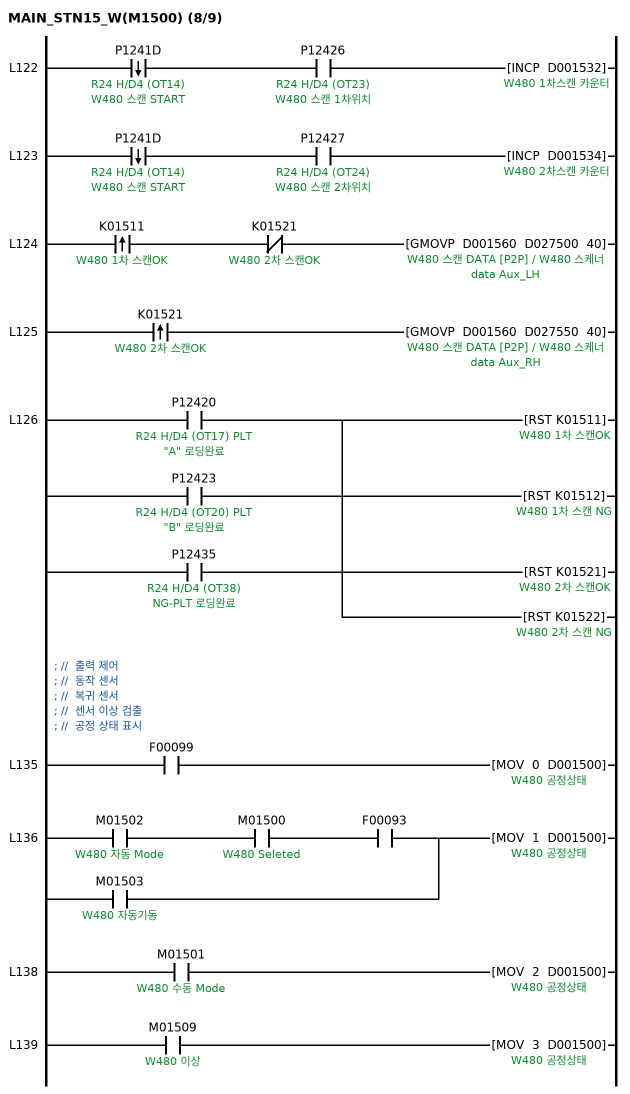
[picture p240: MAIN_STN15_W(M1500) rungs L122-L139]
; L122
LOADN     P1241D	// R24 H/D4 (OT14) W480 스캔 START
AND       P12426	// R24 H/D4 (OT23) W480 스캔 1차위치
INCP      D001532	// W480 1차스캔 카운터
; L123
LOADN     P1241D	// R24 H/D4 (OT14) W480 스캔 START
AND       P12427	// R24 H/D4 (OT24) W480 스캔 2차위치
INCP      D001534	// W480 2차스캔 카운터
; L124
LOADP     K01511	// W480 1차 스캔OK
AND NOT   K01521	// W480 2차 스캔OK
GMOVP     D001560 D027500 40	// W480 스캔 DATA [P2P] / W480 스케너 data Aux_LH
; L125
LOADP     K01521	// W480 2차 스캔OK
GMOVP     D001560 D027550 40	// W480 스캔 DATA [P2P] / W480 스케너 data Aux_RH
; L126
LOAD      P12420	// R24 H/D4 (OT17) PLT "A" 로딩완료
OR        P12423	// R24 H/D4 (OT20) PLT "B" 로딩완료
OR        P12435	// R24 H/D4 (OT38) NG-PLT 로딩완료
RST       K01511	// W480 1차 스캔OK
RST       K01512	// W480 1차 스캔 NG
RST       K01521	// W480 2차 스캔OK
RST       K01522	// W480 2차 스캔 NG
//     //  출력 제어
//   //  동작 센서
//   //  복귀 센서
//     //  센서 이상 검출
//   //  공정 상태 표시
; L135
LOAD      F00099
MOV       0 D001500	// W480 공정상태
; L136
LOAD      M01502	// W480 자동 Mode
AND       M01500	// W480 Seleted
AND       F00093
OR        M01503	// W480 자동기동
MOV       1 D001500	// W480 공정상태
; L138
LOAD      M01501	// W480 수동 Mode
MOV       2 D001500	// W480 공정상태
; L139
LOAD      M01509	// W480 이상
MOV       3 D001500	// W480 공정상태

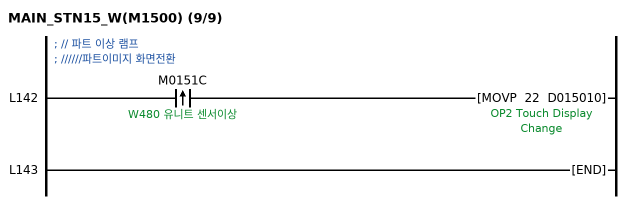
//   // 파트 이상 램프
// //////파트이미지 화면전환
; L142
LOADP     M0151C	// W480 유니트 센서이상
MOVP      22 D015010	// OP2 Touch Display Change
; L143
END

PROGRAM PLT-A (task: 스캔 프로그램)

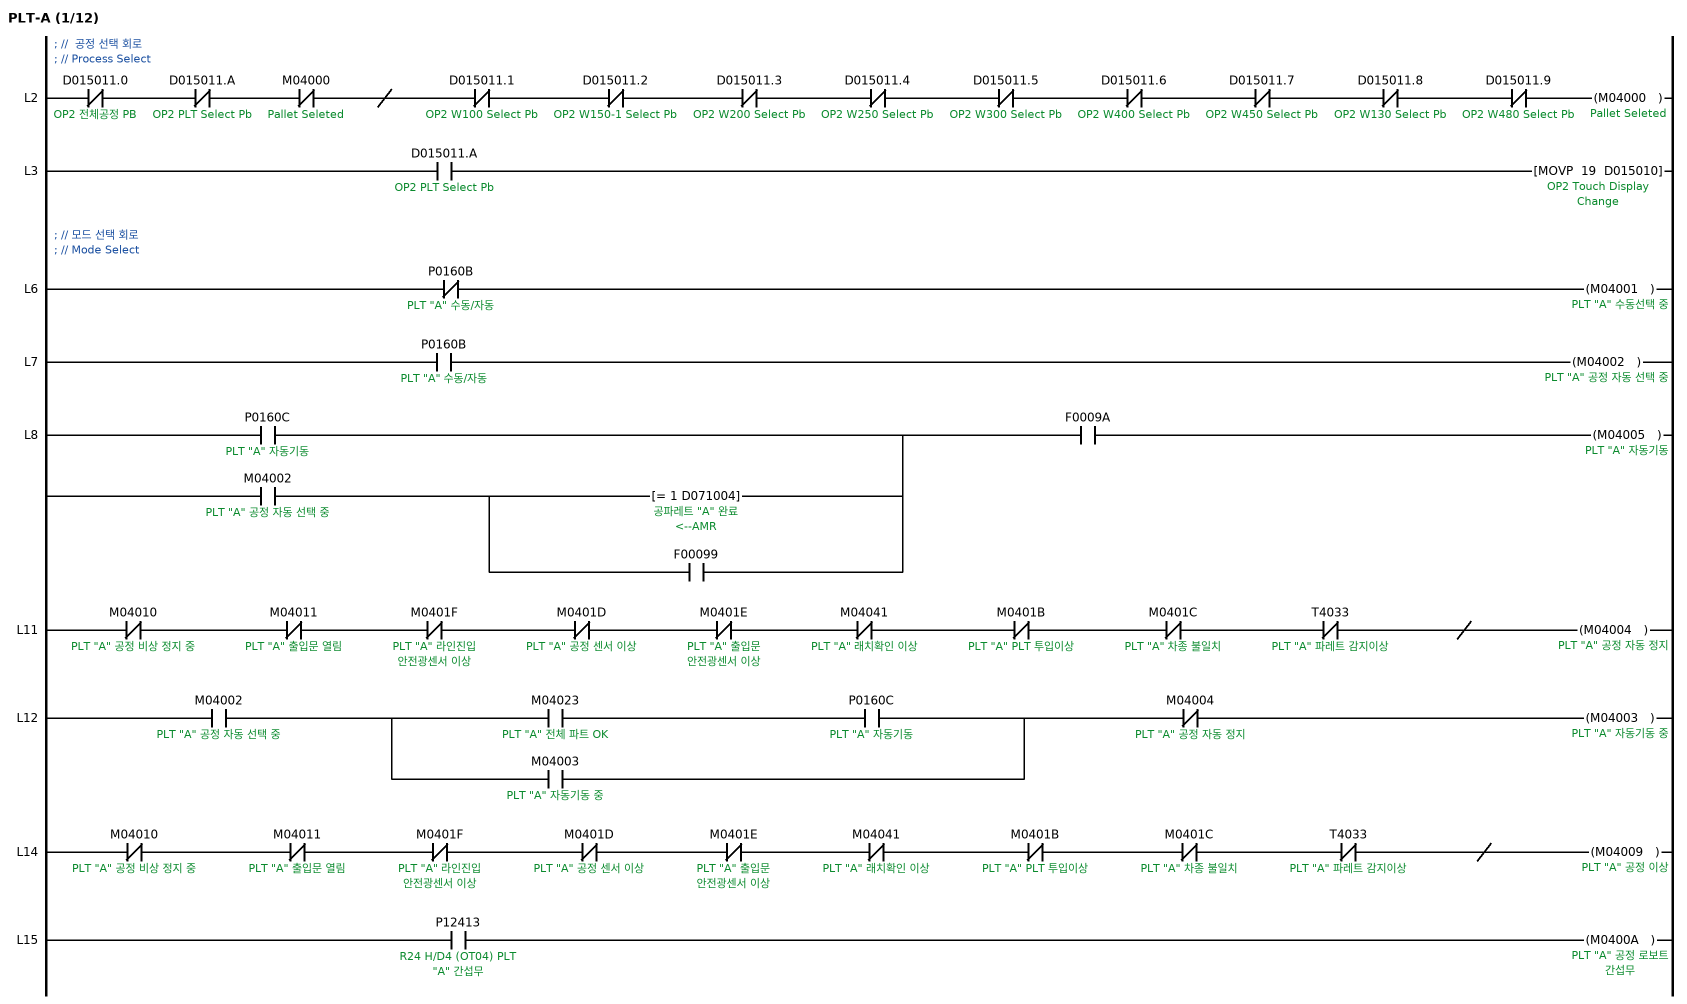
//   //  공정 선택 회로
//   // Process Select
; L2
LOAD NOT  D015011.0	// OP2 전체공정 PB
AND NOT   D015011.A	// OP2 PLT Select Pb
AND NOT   M04000	// Pallet Seleted
NOT
AND NOT   D015011.1	// OP2 W100 Select Pb
AND NOT   D015011.2	// OP2 W150-1 Select Pb
AND NOT   D015011.3	// OP2 W200 Select Pb
AND NOT   D015011.4	// OP2 W250 Select Pb
AND NOT   D015011.5	// OP2 W300 Select Pb
AND NOT   D015011.6	// OP2 W400 Select Pb
AND NOT   D015011.7	// OP2 W450 Select Pb
AND NOT   D015011.8	// OP2 W130 Select Pb
AND NOT   D015011.9	// OP2 W480 Select Pb
OUT       M04000	// Pallet Seleted
; L3
LOAD      D015011.A	// OP2 PLT Select Pb
MOVP      19 D015010	// OP2 Touch Display Change
// // 모드 선택 회로
//   // Mode Select
; L6
LOAD NOT  P0160B	// PLT "A" 수동/자동
OUT       M04001	// PLT "A" 수동선택 중
; L7
LOAD      P0160B	// PLT "A" 수동/자동
OUT       M04002	// PLT "A" 공정 자동 선택 중
; L8
LOAD      P0160C	// PLT "A" 자동기동
LOAD      M04002	// PLT "A" 공정 자동 선택 중
LOAD=     1 D071004	// 공파레트 "A" 완료 <--AMR
OR        F00099
AND LOAD
OR LOAD
AND       F0009A
OUT       M04005	// PLT "A" 자동기동
; L11
LOAD NOT  M04010	// PLT "A" 공정 비상 정지 중
AND NOT   M04011	// PLT "A" 출입문 열림
AND NOT   M0401F	// PLT "A" 라인진입 안전광센서 이상
AND NOT   M0401D	// PLT "A" 공정 센서 이상
AND NOT   M0401E	// PLT "A" 출입문 안전광센서 이상
AND NOT   M04041	// PLT "A" 래치확인 이상
AND NOT   M0401B	// PLT "A" PLT 투입이상
AND NOT   M0401C	// PLT "A" 차종 불일치
AND NOT   T4033	// PLT "A" 파레트 감지이상
NOT
OUT       M04004	// PLT "A" 공정 자동 정지
; L12
LOAD      M04002	// PLT "A" 공정 자동 선택 중
LOAD      M04023	// PLT "A" 전체 파트 OK
AND       P0160C	// PLT "A" 자동기동
OR        M04003	// PLT "A" 자동기동 중
AND LOAD
AND NOT   M04004	// PLT "A" 공정 자동 정지
OUT       M04003	// PLT "A" 자동기동 중
; L14
LOAD NOT  M04010	// PLT "A" 공정 비상 정지 중
AND NOT   M04011	// PLT "A" 출입문 열림
AND NOT   M0401F	// PLT "A" 라인진입 안전광센서 이상
AND NOT   M0401D	// PLT "A" 공정 센서 이상
AND NOT   M0401E	// PLT "A" 출입문 안전광센서 이상
AND NOT   M04041	// PLT "A" 래치확인 이상
AND NOT   M0401B	// PLT "A" PLT 투입이상
AND NOT   M0401C	// PLT "A" 차종 불일치
AND NOT   T4033	// PLT "A" 파레트 감지이상
NOT
OUT       M04009	// PLT "A" 공정 이상
; L15
LOAD      P12413	// R24 H/D4 (OT04) PLT "A" 간섭무
OUT       M0400A	// PLT "A" 공정 로보트 간섭무

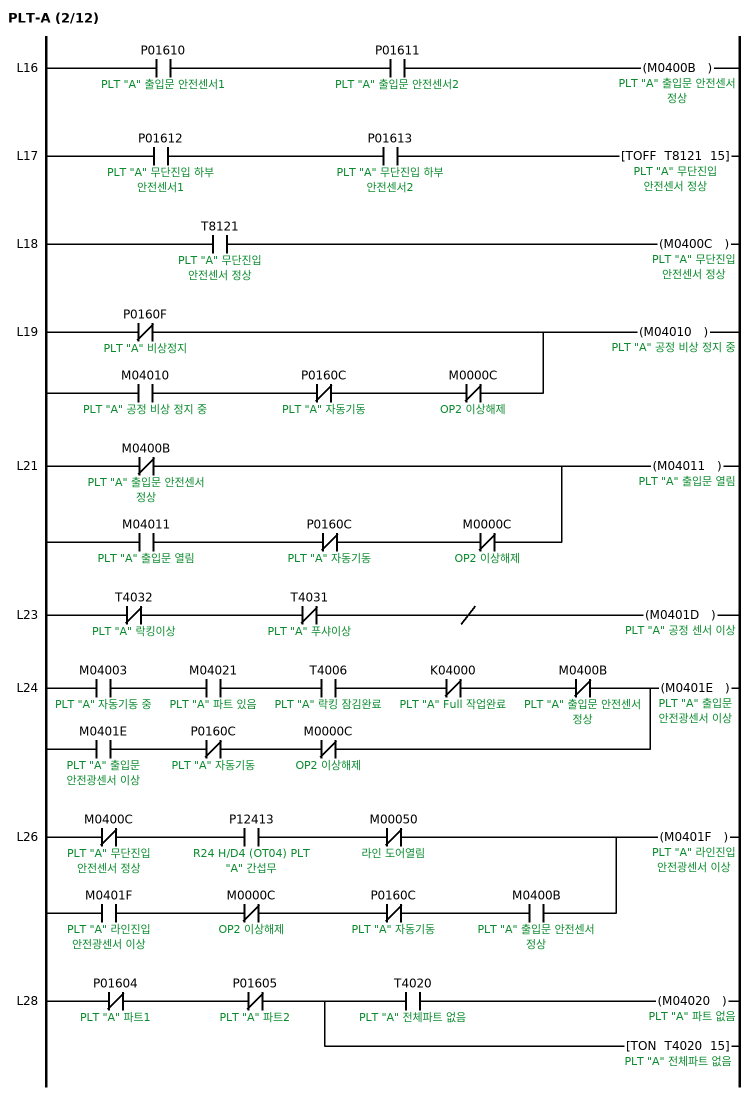
; L16
LOAD      P01610	// PLT "A" 출입문 안전센서1
AND       P01611	// PLT "A" 출입문 안전센서2
OUT       M0400B	// PLT "A" 출입문 안전센서 정상
; L17
LOAD      P01612	// PLT "A" 무단진입 하부 안전센서1
AND       P01613	// PLT "A" 무단진입 하부 안전센서2
TOFF      T8121 15	// PLT "A" 무단진입 안전센서 정상
; L18
LOAD      T8121	// PLT "A" 무단진입 안전센서 정상
OUT       M0400C	// PLT "A" 무단진입 안전센서 정상
; L19
LOAD NOT  P0160F	// PLT "A" 비상정지
LOAD      M04010	// PLT "A" 공정 비상 정지 중
AND NOT   P0160C	// PLT "A" 자동기동
AND NOT   M0000C	// OP2 이상해제
OR LOAD
OUT       M04010	// PLT "A" 공정 비상 정지 중
; L21
LOAD NOT  M0400B	// PLT "A" 출입문 안전센서 정상
LOAD      M04011	// PLT "A" 출입문 열림
AND NOT   P0160C	// PLT "A" 자동기동
AND NOT   M0000C	// OP2 이상해제
OR LOAD
OUT       M04011	// PLT "A" 출입문 열림
; L23
LOAD NOT  T4032	// PLT "A" 락킹이상
AND NOT   T4031	// PLT "A" 푸샤이상
NOT
OUT       M0401D	// PLT "A" 공정 센서 이상
; L24
LOAD      M04003	// PLT "A" 자동기동 중
AND       M04021	// PLT "A" 파트 있음
AND       T4006	// PLT "A" 락킹 잠김완료
AND NOT   K04000	// PLT "A" Full 작업완료
AND NOT   M0400B	// PLT "A" 출입문 안전센서 정상
LOAD      M0401E	// PLT "A" 출입문 안전광센서 이상
AND NOT   P0160C	// PLT "A" 자동기동
AND NOT   M0000C	// OP2 이상해제
OR LOAD
OUT       M0401E	// PLT "A" 출입문 안전광센서 이상
; L26
LOAD NOT  M0400C	// PLT "A" 무단진입 안전센서 정상
AND       P12413	// R24 H/D4 (OT04) PLT "A" 간섭무
AND NOT   M00050	// 라인 도어열림
LOAD      M0401F	// PLT "A" 라인진입 안전광센서 이상
AND NOT   M0000C	// OP2 이상해제
AND NOT   P0160C	// PLT "A" 자동기동
AND       M0400B	// PLT "A" 출입문 안전센서 정상
OR LOAD
OUT       M0401F	// PLT "A" 라인진입 안전광센서 이상
; L28
LOAD NOT  P01604	// PLT "A" 파트1
AND NOT   P01605	// PLT "A" 파트2
MPUSH
AND       T4020	// PLT "A" 전체파트 없음
OUT       M04020	// PLT "A" 파트 없음
MPOP
TON       T4020 15	// PLT "A" 전체파트 없음

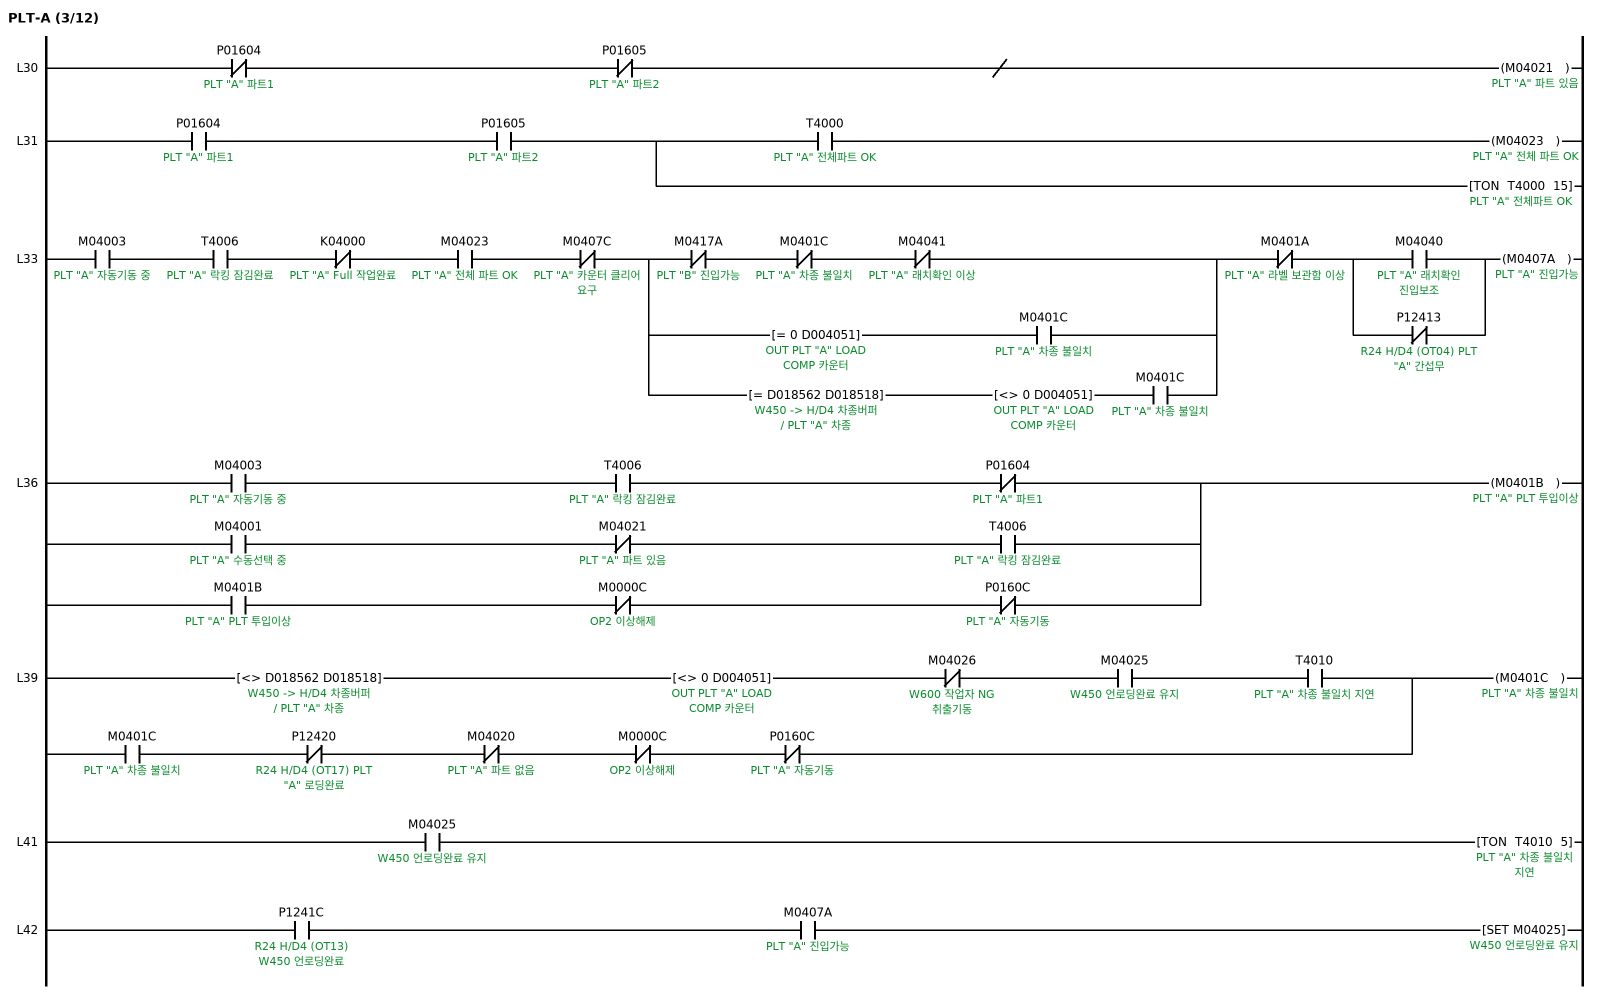
; L30
LOAD NOT  P01604	// PLT "A" 파트1
AND NOT   P01605	// PLT "A" 파트2
NOT
OUT       M04021	// PLT "A" 파트 있음
; L31
LOAD      P01604	// PLT "A" 파트1
AND       P01605	// PLT "A" 파트2
MPUSH
AND       T4000	// PLT "A" 전체파트 OK
OUT       M04023	// PLT "A" 전체 파트 OK
MPOP
TON       T4000 15	// PLT "A" 전체파트 OK
; L33
LOAD      M04003	// PLT "A" 자동기동 중
AND       T4006	// PLT "A" 락킹 잠김완료
AND NOT   K04000	// PLT "A" Full 작업완료
AND       M04023	// PLT "A" 전체 파트 OK
AND NOT   M0407C	// PLT "A" 카운터 클리어 요구
LOAD NOT  M0417A	// PLT "B" 진입가능
AND NOT   M0401C	// PLT "A" 차종 불일치
AND NOT   M04041	// PLT "A" 래치확인 이상
LOAD=     0 D004051	// OUT PLT "A" LOAD COMP 카운터
AND       M0401C	// PLT "A" 차종 불일치
OR LOAD
LOAD=     D018562 D018518	// W450 -> H/D4 차종버퍼 / PLT "A" 차종
AND<>     0 D004051	// OUT PLT "A" LOAD COMP 카운터
AND       M0401C	// PLT "A" 차종 불일치
OR LOAD
AND LOAD
AND NOT   M0401A	// PLT "A" 라벨 보관함 이상
LOAD      M04040	// PLT "A" 래치확인 진입보조
OR NOT    P12413	// R24 H/D4 (OT04) PLT "A" 간섭무
AND LOAD
OUT       M0407A	// PLT "A" 진입가능
; L36
LOAD      M04003	// PLT "A" 자동기동 중
AND       T4006	// PLT "A" 락킹 잠김완료
AND NOT   P01604	// PLT "A" 파트1
LOAD      M04001	// PLT "A" 수동선택 중
AND NOT   M04021	// PLT "A" 파트 있음
AND       T4006	// PLT "A" 락킹 잠김완료
OR LOAD
LOAD      M0401B	// PLT "A" PLT 투입이상
AND NOT   M0000C	// OP2 이상해제
AND NOT   P0160C	// PLT "A" 자동기동
OR LOAD
OUT       M0401B	// PLT "A" PLT 투입이상
; L39
LOAD<>    D018562 D018518	// W450 -> H/D4 차종버퍼 / PLT "A" 차종
AND<>     0 D004051	// OUT PLT "A" LOAD COMP 카운터
AND NOT   M04026	// W600 작업자 NG 취출기동
AND       M04025	// W450 언로딩완료 유지
AND       T4010	// PLT "A" 차종 불일치 지연
LOAD      M0401C	// PLT "A" 차종 불일치
AND NOT   P12420	// R24 H/D4 (OT17) PLT "A" 로딩완료
AND NOT   M04020	// PLT "A" 파트 없음
AND NOT   M0000C	// OP2 이상해제
AND NOT   P0160C	// PLT "A" 자동기동
OR LOAD
OUT       M0401C	// PLT "A" 차종 불일치
; L41
LOAD      M04025	// W450 언로딩완료 유지
TON       T4010 5	// PLT "A" 차종 불일치 지연
; L42
LOAD      P1241C	// R24 H/D4 (OT13) W450 언로딩완료
AND       M0407A	// PLT "A" 진입가능
SET       M04025	// W450 언로딩완료 유지

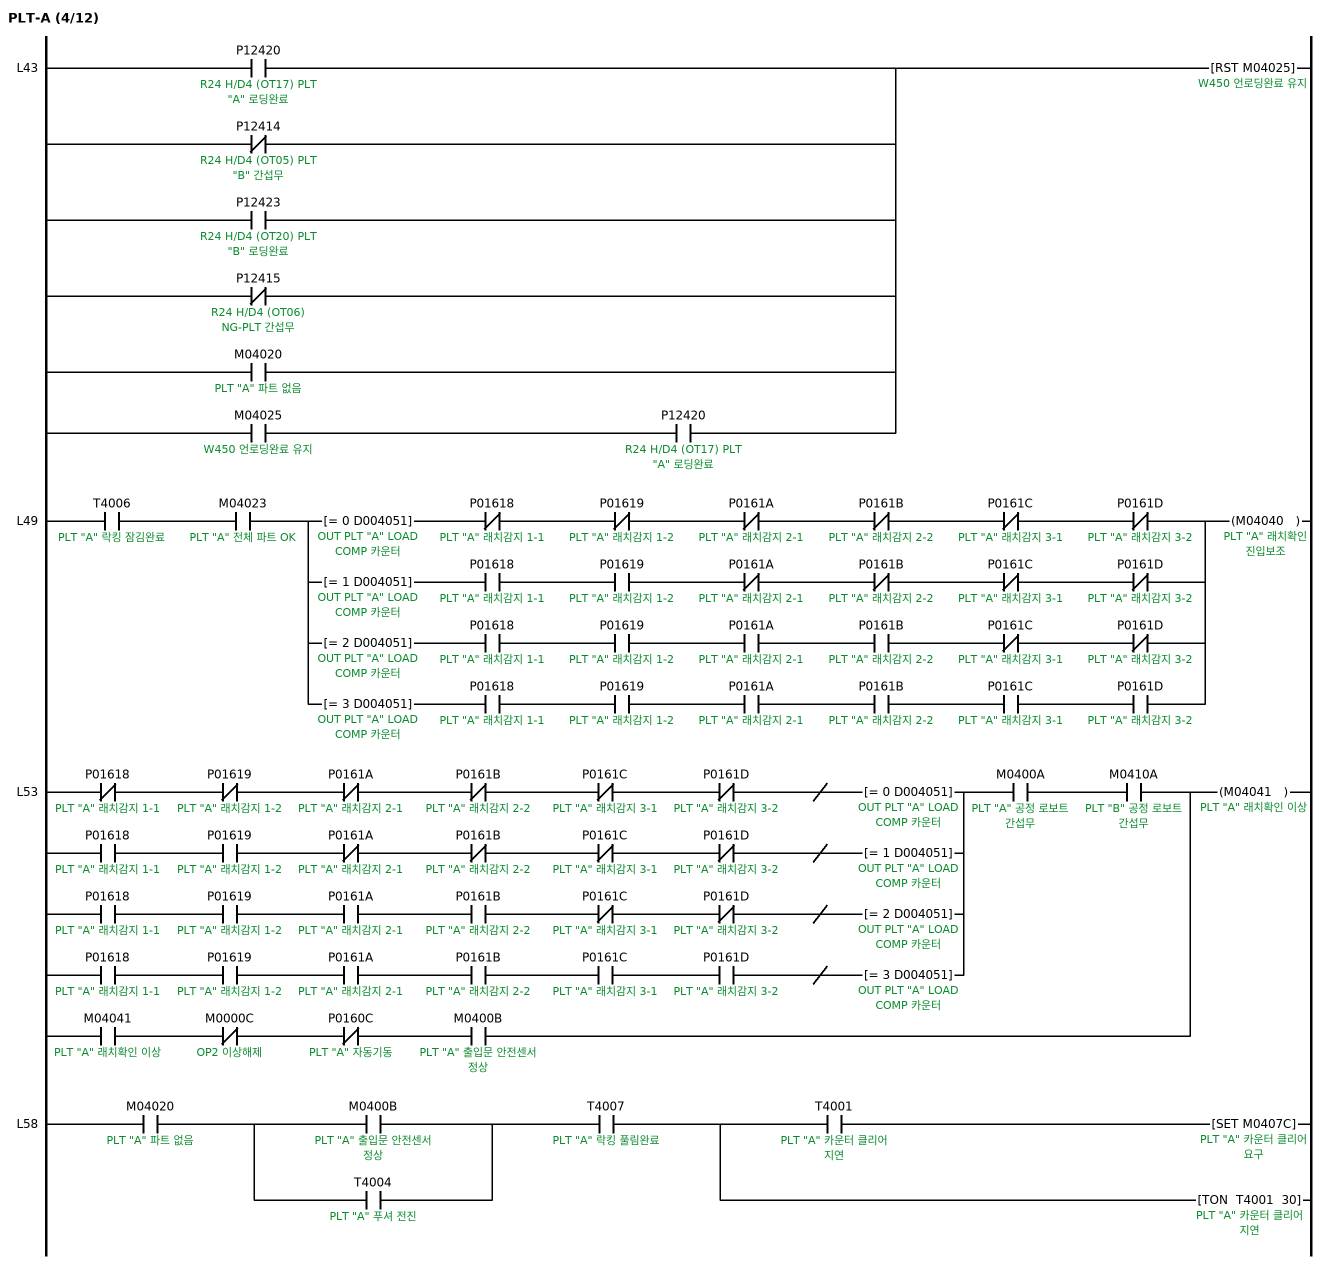
; L43
LOAD      P12420	// R24 H/D4 (OT17) PLT "A" 로딩완료
OR NOT    P12414	// R24 H/D4 (OT05) PLT "B" 간섭무
OR        P12423	// R24 H/D4 (OT20) PLT "B" 로딩완료
OR NOT    P12415	// R24 H/D4 (OT06) NG-PLT 간섭무
OR        M04020	// PLT "A" 파트 없음
LOAD      M04025	// W450 언로딩완료 유지
AND       P12420	// R24 H/D4 (OT17) PLT "A" 로딩완료
OR LOAD
RST       M04025	// W450 언로딩완료 유지
; L49
LOAD      T4006	// PLT "A" 락킹 잠김완료
AND       M04023	// PLT "A" 전체 파트 OK
LOAD=     0 D004051	// OUT PLT "A" LOAD COMP 카운터
AND NOT   P01618	// PLT "A" 래치감지 1-1
AND NOT   P01619	// PLT "A" 래치감지 1-2
AND NOT   P0161A	// PLT "A" 래치감지 2-1
AND NOT   P0161B	// PLT "A" 래치감지 2-2
AND NOT   P0161C	// PLT "A" 래치감지 3-1
AND NOT   P0161D	// PLT "A" 래치감지 3-2
LOAD=     1 D004051	// OUT PLT "A" LOAD COMP 카운터
AND       P01618	// PLT "A" 래치감지 1-1
AND       P01619	// PLT "A" 래치감지 1-2
AND NOT   P0161A	// PLT "A" 래치감지 2-1
AND NOT   P0161B	// PLT "A" 래치감지 2-2
AND NOT   P0161C	// PLT "A" 래치감지 3-1
AND NOT   P0161D	// PLT "A" 래치감지 3-2
OR LOAD
LOAD=     2 D004051	// OUT PLT "A" LOAD COMP 카운터
AND       P01618	// PLT "A" 래치감지 1-1
AND       P01619	// PLT "A" 래치감지 1-2
AND       P0161A	// PLT "A" 래치감지 2-1
AND       P0161B	// PLT "A" 래치감지 2-2
AND NOT   P0161C	// PLT "A" 래치감지 3-1
AND NOT   P0161D	// PLT "A" 래치감지 3-2
OR LOAD
LOAD=     3 D004051	// OUT PLT "A" LOAD COMP 카운터
AND       P01618	// PLT "A" 래치감지 1-1
AND       P01619	// PLT "A" 래치감지 1-2
AND       P0161A	// PLT "A" 래치감지 2-1
AND       P0161B	// PLT "A" 래치감지 2-2
AND       P0161C	// PLT "A" 래치감지 3-1
AND       P0161D	// PLT "A" 래치감지 3-2
OR LOAD
AND LOAD
OUT       M04040	// PLT "A" 래치확인 진입보조
; L53
LOAD NOT  P01618	// PLT "A" 래치감지 1-1
AND NOT   P01619	// PLT "A" 래치감지 1-2
AND NOT   P0161A	// PLT "A" 래치감지 2-1
AND NOT   P0161B	// PLT "A" 래치감지 2-2
AND NOT   P0161C	// PLT "A" 래치감지 3-1
AND NOT   P0161D	// PLT "A" 래치감지 3-2
NOT
AND=      0 D004051	// OUT PLT "A" LOAD COMP 카운터
LOAD      P01618	// PLT "A" 래치감지 1-1
AND       P01619	// PLT "A" 래치감지 1-2
AND NOT   P0161A	// PLT "A" 래치감지 2-1
AND NOT   P0161B	// PLT "A" 래치감지 2-2
AND NOT   P0161C	// PLT "A" 래치감지 3-1
AND NOT   P0161D	// PLT "A" 래치감지 3-2
NOT
AND=      1 D004051	// OUT PLT "A" LOAD COMP 카운터
OR LOAD
LOAD      P01618	// PLT "A" 래치감지 1-1
AND       P01619	// PLT "A" 래치감지 1-2
AND       P0161A	// PLT "A" 래치감지 2-1
AND       P0161B	// PLT "A" 래치감지 2-2
AND NOT   P0161C	// PLT "A" 래치감지 3-1
AND NOT   P0161D	// PLT "A" 래치감지 3-2
NOT
AND=      2 D004051	// OUT PLT "A" LOAD COMP 카운터
OR LOAD
LOAD      P01618	// PLT "A" 래치감지 1-1
AND       P01619	// PLT "A" 래치감지 1-2
AND       P0161A	// PLT "A" 래치감지 2-1
AND       P0161B	// PLT "A" 래치감지 2-2
AND       P0161C	// PLT "A" 래치감지 3-1
AND       P0161D	// PLT "A" 래치감지 3-2
NOT
AND=      3 D004051	// OUT PLT "A" LOAD COMP 카운터
OR LOAD
AND       M0400A	// PLT "A" 공정 로보트 간섭무
AND       M0410A	// PLT "B" 공정 로보트 간섭무
LOAD      M04041	// PLT "A" 래치확인 이상
AND NOT   M0000C	// OP2 이상해제
AND NOT   P0160C	// PLT "A" 자동기동
AND       M0400B	// PLT "A" 출입문 안전센서 정상
OR LOAD
OUT       M04041	// PLT "A" 래치확인 이상
; L58
LOAD      M04020	// PLT "A" 파트 없음
LOAD      M0400B	// PLT "A" 출입문 안전센서 정상
OR        T4004	// PLT "A" 푸셔 전진
AND LOAD
AND       T4007	// PLT "A" 락킹 풀림완료
MPUSH
AND       T4001	// PLT "A" 카운터 클리어 지연
SET       M0407C	// PLT "A" 카운터 클리어 요구
MPOP
TON       T4001 30	// PLT "A" 카운터 클리어 지연

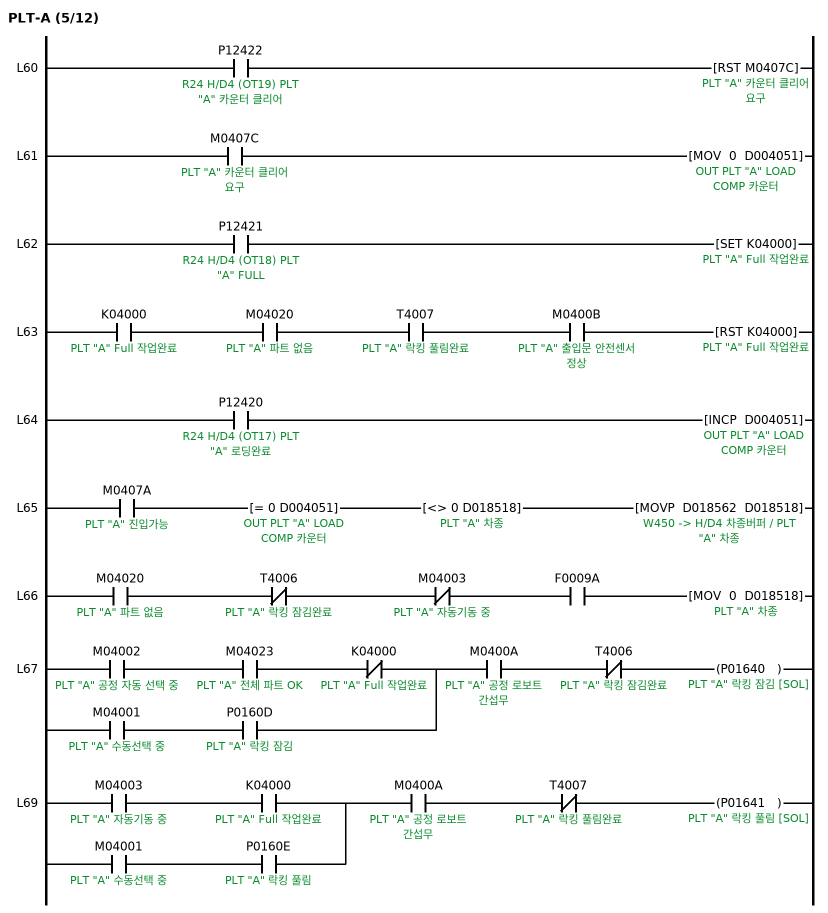
; L60
LOAD      P12422	// R24 H/D4 (OT19) PLT "A" 카운터 클리어
RST       M0407C	// PLT "A" 카운터 클리어 요구
; L61
LOAD      M0407C	// PLT "A" 카운터 클리어 요구
MOV       0 D004051	// OUT PLT "A" LOAD COMP 카운터
; L62
LOAD      P12421	// R24 H/D4 (OT18) PLT "A" FULL
SET       K04000	// PLT "A" Full 작업완료
; L63
LOAD      K04000	// PLT "A" Full 작업완료
AND       M04020	// PLT "A" 파트 없음
AND       T4007	// PLT "A" 락킹 풀림완료
AND       M0400B	// PLT "A" 출입문 안전센서 정상
RST       K04000	// PLT "A" Full 작업완료
; L64
LOAD      P12420	// R24 H/D4 (OT17) PLT "A" 로딩완료
INCP      D004051	// OUT PLT "A" LOAD COMP 카운터
; L65
LOAD      M0407A	// PLT "A" 진입가능
AND=      0 D004051	// OUT PLT "A" LOAD COMP 카운터
AND<>     0 D018518	// PLT "A" 차종
MOVP      D018562 D018518	// W450 -> H/D4 차종버퍼 / PLT "A" 차종
; L66
LOAD      M04020	// PLT "A" 파트 없음
AND NOT   T4006	// PLT "A" 락킹 잠김완료
AND NOT   M04003	// PLT "A" 자동기동 중
AND       F0009A
MOV       0 D018518	// PLT "A" 차종
; L67
LOAD      M04002	// PLT "A" 공정 자동 선택 중
AND       M04023	// PLT "A" 전체 파트 OK
AND NOT   K04000	// PLT "A" Full 작업완료
LOAD      M04001	// PLT "A" 수동선택 중
AND       P0160D	// PLT "A" 락킹 잠김
OR LOAD
AND       M0400A	// PLT "A" 공정 로보트 간섭무
AND NOT   T4006	// PLT "A" 락킹 잠김완료
OUT       P01640	// PLT "A" 락킹 잠김 [SOL]
; L69
LOAD      M04003	// PLT "A" 자동기동 중
AND       K04000	// PLT "A" Full 작업완료
LOAD      M04001	// PLT "A" 수동선택 중
AND       P0160E	// PLT "A" 락킹 풀림
OR LOAD
AND       M0400A	// PLT "A" 공정 로보트 간섭무
AND NOT   T4007	// PLT "A" 락킹 풀림완료
OUT       P01641	// PLT "A" 락킹 풀림 [SOL]

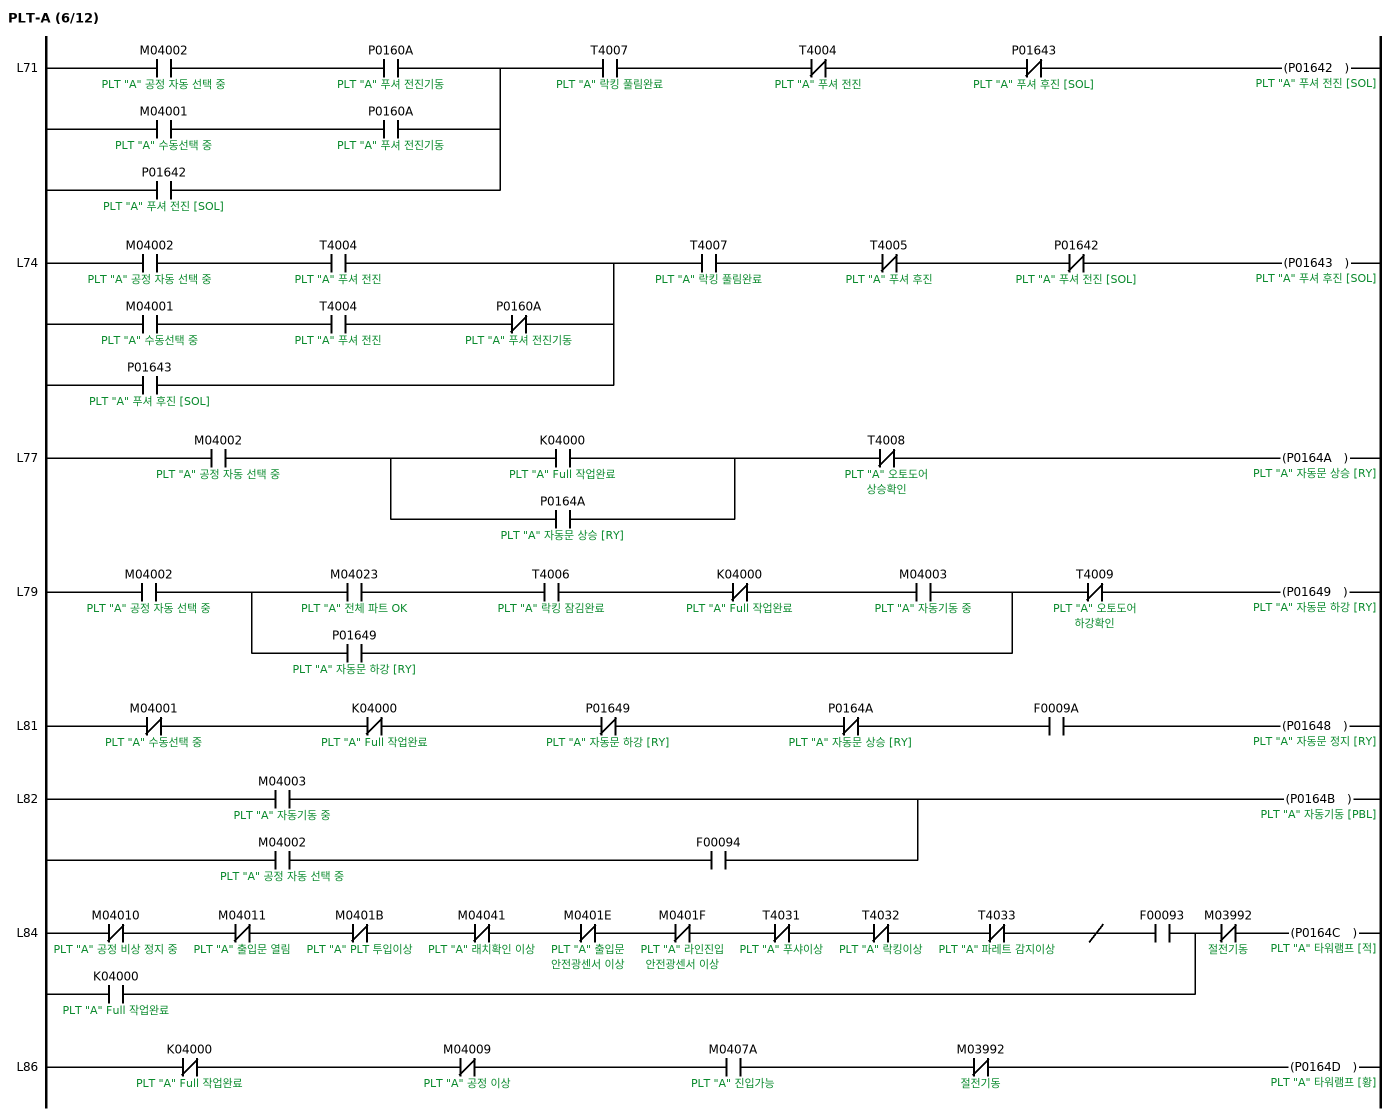
; L71
LOAD      M04002	// PLT "A" 공정 자동 선택 중
AND       P0160A	// PLT "A" 푸셔 전진기동
LOAD      M04001	// PLT "A" 수동선택 중
AND       P0160A	// PLT "A" 푸셔 전진기동
OR LOAD
OR        P01642	// PLT "A" 푸셔 전진 [SOL]
AND       T4007	// PLT "A" 락킹 풀림완료
AND NOT   T4004	// PLT "A" 푸셔 전진
AND NOT   P01643	// PLT "A" 푸셔 후진 [SOL]
OUT       P01642	// PLT "A" 푸셔 전진 [SOL]
; L74
LOAD      M04002	// PLT "A" 공정 자동 선택 중
AND       T4004	// PLT "A" 푸셔 전진
LOAD      M04001	// PLT "A" 수동선택 중
AND       T4004	// PLT "A" 푸셔 전진
AND NOT   P0160A	// PLT "A" 푸셔 전진기동
OR LOAD
OR        P01643	// PLT "A" 푸셔 후진 [SOL]
AND       T4007	// PLT "A" 락킹 풀림완료
AND NOT   T4005	// PLT "A" 푸셔 후진
AND NOT   P01642	// PLT "A" 푸셔 전진 [SOL]
OUT       P01643	// PLT "A" 푸셔 후진 [SOL]
; L77
LOAD      M04002	// PLT "A" 공정 자동 선택 중
LOAD      K04000	// PLT "A" Full 작업완료
OR        P0164A	// PLT "A" 자동문 상승 [RY]
AND LOAD
AND NOT   T4008	// PLT "A" 오토도어 상승확인
OUT       P0164A	// PLT "A" 자동문 상승 [RY]
; L79
LOAD      M04002	// PLT "A" 공정 자동 선택 중
LOAD      M04023	// PLT "A" 전체 파트 OK
AND       T4006	// PLT "A" 락킹 잠김완료
AND NOT   K04000	// PLT "A" Full 작업완료
AND       M04003	// PLT "A" 자동기동 중
OR        P01649	// PLT "A" 자동문 하강 [RY]
AND LOAD
AND NOT   T4009	// PLT "A" 오토도어 하강확인
OUT       P01649	// PLT "A" 자동문 하강 [RY]
; L81
LOAD NOT  M04001	// PLT "A" 수동선택 중
AND NOT   K04000	// PLT "A" Full 작업완료
AND NOT   P01649	// PLT "A" 자동문 하강 [RY]
AND NOT   P0164A	// PLT "A" 자동문 상승 [RY]
AND       F0009A
OUT       P01648	// PLT "A" 자동문 정지 [RY]
; L82
LOAD      M04003	// PLT "A" 자동기동 중
LOAD      M04002	// PLT "A" 공정 자동 선택 중
AND       F00094
OR LOAD
OUT       P0164B	// PLT "A" 자동기동 [PBL]
; L84
LOAD NOT  M04010	// PLT "A" 공정 비상 정지 중
AND NOT   M04011	// PLT "A" 출입문 열림
AND NOT   M0401B	// PLT "A" PLT 투입이상
AND NOT   M04041	// PLT "A" 래치확인 이상
AND NOT   M0401E	// PLT "A" 출입문 안전광센서 이상
AND NOT   M0401F	// PLT "A" 라인진입 안전광센서 이상
AND NOT   T4031	// PLT "A" 푸샤이상
AND NOT   T4032	// PLT "A" 락킹이상
AND NOT   T4033	// PLT "A" 파레트 감지이상
NOT
AND       F00093
OR        K04000	// PLT "A" Full 작업완료
AND NOT   M03992	// 절전기동
OUT       P0164C	// PLT "A" 타워램프 [적]
; L86
LOAD NOT  K04000	// PLT "A" Full 작업완료
AND NOT   M04009	// PLT "A" 공정 이상
AND       M0407A	// PLT "A" 진입가능
AND NOT   M03992	// 절전기동
OUT       P0164D	// PLT "A" 타워램프 [황]

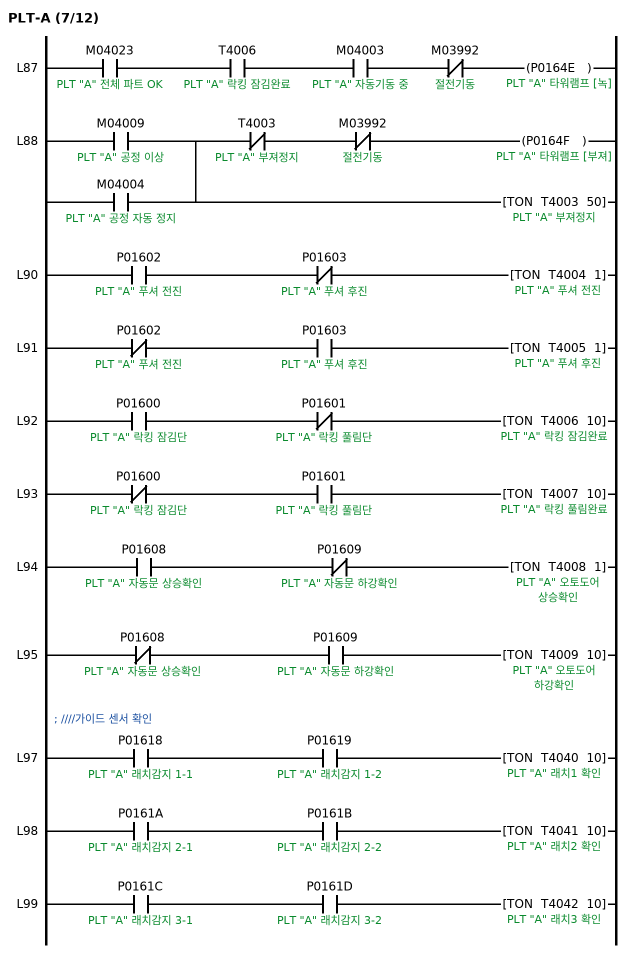
; L87
LOAD      M04023	// PLT "A" 전체 파트 OK
AND       T4006	// PLT "A" 락킹 잠김완료
AND       M04003	// PLT "A" 자동기동 중
AND NOT   M03992	// 절전기동
OUT       P0164E	// PLT "A" 타워램프 [녹]
; L88
LOAD      M04009	// PLT "A" 공정 이상
OR        M04004	// PLT "A" 공정 자동 정지
MPUSH
AND NOT   T4003	// PLT "A" 부져정지
AND NOT   M03992	// 절전기동
OUT       P0164F	// PLT "A" 타워램프 [부져]
MPOP
TON       T4003 50	// PLT "A" 부져정지
; L90
LOAD      P01602	// PLT "A" 푸셔 전진
AND NOT   P01603	// PLT "A" 푸셔 후진
TON       T4004 1	// PLT "A" 푸셔 전진
; L91
LOAD NOT  P01602	// PLT "A" 푸셔 전진
AND       P01603	// PLT "A" 푸셔 후진
TON       T4005 1	// PLT "A" 푸셔 후진
; L92
LOAD      P01600	// PLT "A" 락킹 잠김단
AND NOT   P01601	// PLT "A" 락킹 풀림단
TON       T4006 10	// PLT "A" 락킹 잠김완료
; L93
LOAD NOT  P01600	// PLT "A" 락킹 잠김단
AND       P01601	// PLT "A" 락킹 풀림단
TON       T4007 10	// PLT "A" 락킹 풀림완료
; L94
LOAD      P01608	// PLT "A" 자동문 상승확인
AND NOT   P01609	// PLT "A" 자동문 하강확인
TON       T4008 1	// PLT "A" 오토도어 상승확인
; L95
LOAD NOT  P01608	// PLT "A" 자동문 상승확인
AND       P01609	// PLT "A" 자동문 하강확인
TON       T4009 10	// PLT "A" 오토도어 하강확인
// ////가이드 센서 확인
; L97
LOAD      P01618	// PLT "A" 래치감지 1-1
AND       P01619	// PLT "A" 래치감지 1-2
TON       T4040 10	// PLT "A" 래치1 확인
; L98
LOAD      P0161A	// PLT "A" 래치감지 2-1
AND       P0161B	// PLT "A" 래치감지 2-2
TON       T4041 10	// PLT "A" 래치2 확인
; L99
LOAD      P0161C	// PLT "A" 래치감지 3-1
AND       P0161D	// PLT "A" 래치감지 3-2
TON       T4042 10	// PLT "A" 래치3 확인

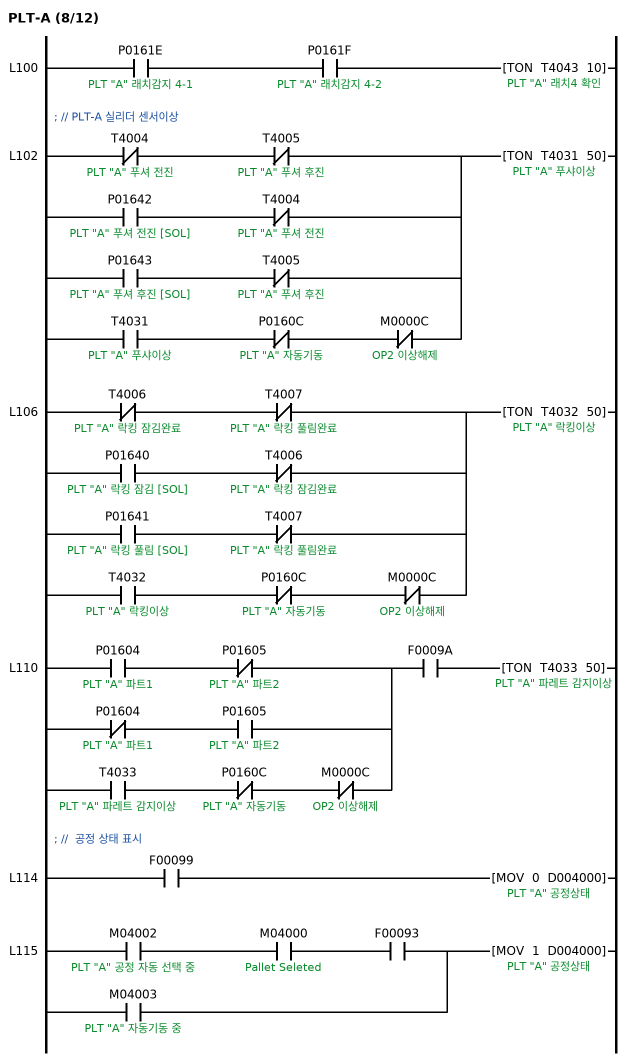
; L100
LOAD      P0161E	// PLT "A" 래치감지 4-1
AND       P0161F	// PLT "A" 래치감지 4-2
TON       T4043 10	// PLT "A" 래치4 확인
// // PLT-A 실리더 센서이상
; L102
LOAD NOT  T4004	// PLT "A" 푸셔 전진
AND NOT   T4005	// PLT "A" 푸셔 후진
LOAD      P01642	// PLT "A" 푸셔 전진 [SOL]
AND NOT   T4004	// PLT "A" 푸셔 전진
OR LOAD
LOAD      P01643	// PLT "A" 푸셔 후진 [SOL]
AND NOT   T4005	// PLT "A" 푸셔 후진
OR LOAD
LOAD      T4031	// PLT "A" 푸샤이상
AND NOT   P0160C	// PLT "A" 자동기동
AND NOT   M0000C	// OP2 이상해제
OR LOAD
TON       T4031 50	// PLT "A" 푸샤이상
; L106
LOAD NOT  T4006	// PLT "A" 락킹 잠김완료
AND NOT   T4007	// PLT "A" 락킹 풀림완료
LOAD      P01640	// PLT "A" 락킹 잠김 [SOL]
AND NOT   T4006	// PLT "A" 락킹 잠김완료
OR LOAD
LOAD      P01641	// PLT "A" 락킹 풀림 [SOL]
AND NOT   T4007	// PLT "A" 락킹 풀림완료
OR LOAD
LOAD      T4032	// PLT "A" 락킹이상
AND NOT   P0160C	// PLT "A" 자동기동
AND NOT   M0000C	// OP2 이상해제
OR LOAD
TON       T4032 50	// PLT "A" 락킹이상
; L110
LOAD      P01604	// PLT "A" 파트1
AND NOT   P01605	// PLT "A" 파트2
LOAD NOT  P01604	// PLT "A" 파트1
AND       P01605	// PLT "A" 파트2
OR LOAD
LOAD      T4033	// PLT "A" 파레트 감지이상
AND NOT   P0160C	// PLT "A" 자동기동
AND NOT   M0000C	// OP2 이상해제
OR LOAD
AND       F0009A
TON       T4033 50	// PLT "A" 파레트 감지이상
//   //  공정 상태 표시
; L114
LOAD      F00099
MOV       0 D004000	// PLT "A" 공정상태
; L115
LOAD      M04002	// PLT "A" 공정 자동 선택 중
AND       M04000	// Pallet Seleted
AND       F00093
OR        M04003	// PLT "A" 자동기동 중
MOV       1 D004000	// PLT "A" 공정상태

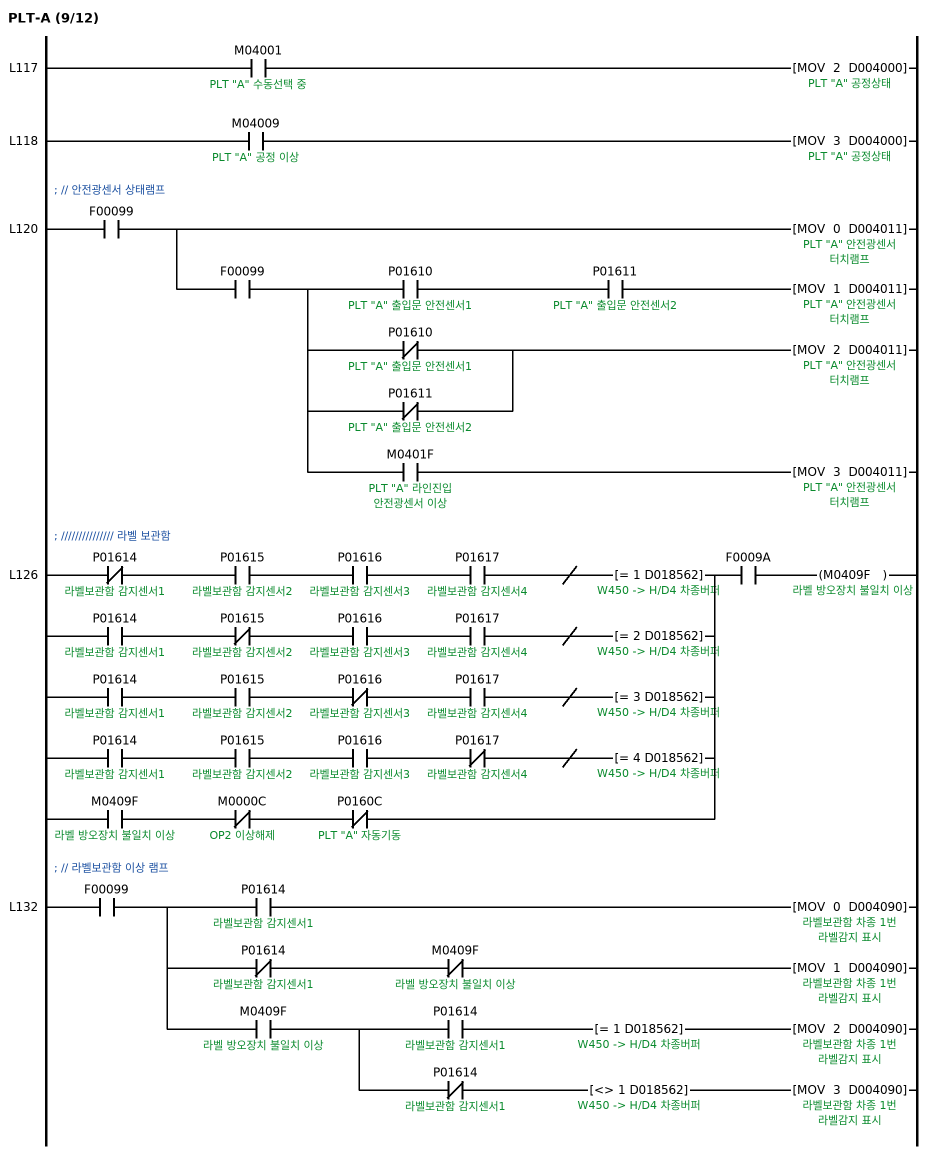
; L117
LOAD      M04001	// PLT "A" 수동선택 중
MOV       2 D004000	// PLT "A" 공정상태
; L118
LOAD      M04009	// PLT "A" 공정 이상
MOV       3 D004000	// PLT "A" 공정상태
//   // 안전광센서 상태램프
; L120
LOAD      F00099
MOV       0 D004011	// PLT "A" 안전광센서 터치램프
AND       F00099
MPUSH
AND       P01610	// PLT "A" 출입문 안전센서1
AND       P01611	// PLT "A" 출입문 안전센서2
MOV       1 D004011	// PLT "A" 안전광센서 터치램프
MLOAD
LOAD NOT  P01610	// PLT "A" 출입문 안전센서1
OR NOT    P01611	// PLT "A" 출입문 안전센서2
AND LOAD
MOV       2 D004011	// PLT "A" 안전광센서 터치램프
MPOP
AND       M0401F	// PLT "A" 라인진입 안전광센서 이상
MOV       3 D004011	// PLT "A" 안전광센서 터치램프
// /////////////// 라벨 보관함
; L126
LOAD NOT  P01614	// 라벨보관함 감지센서1
AND       P01615	// 라벨보관함 감지센서2
AND       P01616	// 라벨보관함 감지센서3
AND       P01617	// 라벨보관함 감지센서4
NOT
AND=      1 D018562	// W450 -> H/D4 차종버퍼
LOAD      P01614	// 라벨보관함 감지센서1
AND NOT   P01615	// 라벨보관함 감지센서2
AND       P01616	// 라벨보관함 감지센서3
AND       P01617	// 라벨보관함 감지센서4
NOT
AND=      2 D018562	// W450 -> H/D4 차종버퍼
OR LOAD
LOAD      P01614	// 라벨보관함 감지센서1
AND       P01615	// 라벨보관함 감지센서2
AND NOT   P01616	// 라벨보관함 감지센서3
AND       P01617	// 라벨보관함 감지센서4
NOT
AND=      3 D018562	// W450 -> H/D4 차종버퍼
OR LOAD
LOAD      P01614	// 라벨보관함 감지센서1
AND       P01615	// 라벨보관함 감지센서2
AND       P01616	// 라벨보관함 감지센서3
AND NOT   P01617	// 라벨보관함 감지센서4
NOT
AND=      4 D018562	// W450 -> H/D4 차종버퍼
OR LOAD
LOAD      M0409F	// 라벨 방오장치 불일치 이상
AND NOT   M0000C	// OP2 이상해제
AND NOT   P0160C	// PLT "A" 자동기동
OR LOAD
AND       F0009A
OUT       M0409F	// 라벨 방오장치 불일치 이상
//   // 라벨보관함 이상 램프
; L132
LOAD      F00099
MPUSH
AND       P01614	// 라벨보관함 감지센서1
MOV       0 D004090	// 라벨보관함 차종 1번 라벨감지 표시
MLOAD
AND NOT   P01614	// 라벨보관함 감지센서1
AND NOT   M0409F	// 라벨 방오장치 불일치 이상
MOV       1 D004090	// 라벨보관함 차종 1번 라벨감지 표시
MPOP
AND       M0409F	// 라벨 방오장치 불일치 이상
MPUSH
AND       P01614	// 라벨보관함 감지센서1
AND=      1 D018562	// W450 -> H/D4 차종버퍼
MOV       2 D004090	// 라벨보관함 차종 1번 라벨감지 표시
MPOP
AND NOT   P01614	// 라벨보관함 감지센서1
AND<>     1 D018562	// W450 -> H/D4 차종버퍼
MOV       3 D004090	// 라벨보관함 차종 1번 라벨감지 표시

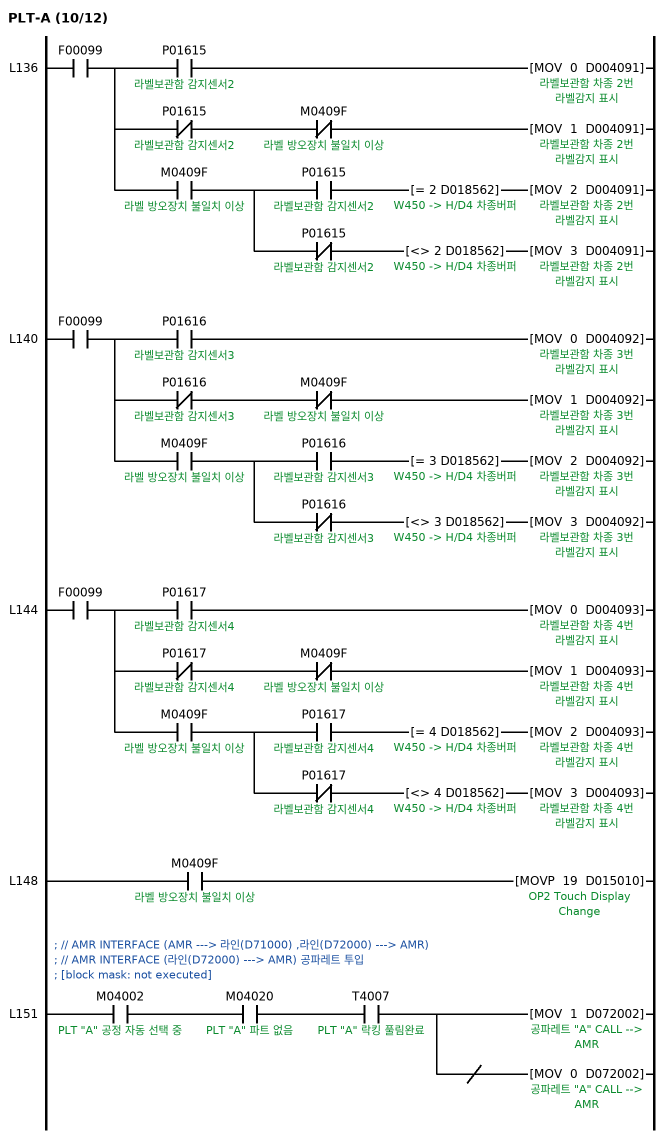
; L136
LOAD      F00099
MPUSH
AND       P01615	// 라벨보관함 감지센서2
MOV       0 D004091	// 라벨보관함 차종 2번 라벨감지 표시
MLOAD
AND NOT   P01615	// 라벨보관함 감지센서2
AND NOT   M0409F	// 라벨 방오장치 불일치 이상
MOV       1 D004091	// 라벨보관함 차종 2번 라벨감지 표시
MPOP
AND       M0409F	// 라벨 방오장치 불일치 이상
MPUSH
AND       P01615	// 라벨보관함 감지센서2
AND=      2 D018562	// W450 -> H/D4 차종버퍼
MOV       2 D004091	// 라벨보관함 차종 2번 라벨감지 표시
MPOP
AND NOT   P01615	// 라벨보관함 감지센서2
AND<>     2 D018562	// W450 -> H/D4 차종버퍼
MOV       3 D004091	// 라벨보관함 차종 2번 라벨감지 표시
; L140
LOAD      F00099
MPUSH
AND       P01616	// 라벨보관함 감지센서3
MOV       0 D004092	// 라벨보관함 차종 3번 라벨감지 표시
MLOAD
AND NOT   P01616	// 라벨보관함 감지센서3
AND NOT   M0409F	// 라벨 방오장치 불일치 이상
MOV       1 D004092	// 라벨보관함 차종 3번 라벨감지 표시
MPOP
AND       M0409F	// 라벨 방오장치 불일치 이상
MPUSH
AND       P01616	// 라벨보관함 감지센서3
AND=      3 D018562	// W450 -> H/D4 차종버퍼
MOV       2 D004092	// 라벨보관함 차종 3번 라벨감지 표시
MPOP
AND NOT   P01616	// 라벨보관함 감지센서3
AND<>     3 D018562	// W450 -> H/D4 차종버퍼
MOV       3 D004092	// 라벨보관함 차종 3번 라벨감지 표시
; L144
LOAD      F00099
MPUSH
AND       P01617	// 라벨보관함 감지센서4
MOV       0 D004093	// 라벨보관함 차종 4번 라벨감지 표시
MLOAD
AND NOT   P01617	// 라벨보관함 감지센서4
AND NOT   M0409F	// 라벨 방오장치 불일치 이상
MOV       1 D004093	// 라벨보관함 차종 4번 라벨감지 표시
MPOP
AND       M0409F	// 라벨 방오장치 불일치 이상
MPUSH
AND       P01617	// 라벨보관함 감지센서4
AND=      4 D018562	// W450 -> H/D4 차종버퍼
MOV       2 D004093	// 라벨보관함 차종 4번 라벨감지 표시
MPOP
AND NOT   P01617	// 라벨보관함 감지센서4
AND<>     4 D018562	// W450 -> H/D4 차종버퍼
MOV       3 D004093	// 라벨보관함 차종 4번 라벨감지 표시
; L148
LOAD      M0409F	// 라벨 방오장치 불일치 이상
MOVP      19 D015010	// OP2 Touch Display Change
//   // AMR INTERFACE (AMR ---> 라인(D71000) ,라인(D72000) ---> AMR)
//   // AMR INTERFACE (라인(D72000) ---> AMR) 공파레트 투입
; L151 (block mask: not executed)
LOAD      M04002	// PLT "A" 공정 자동 선택 중
AND       M04020	// PLT "A" 파트 없음
AND       T4007	// PLT "A" 락킹 풀림완료
MOV       1 D072002	// 공파레트 "A" CALL --> AMR
NOT
MOV       0 D072002	// 공파레트 "A" CALL --> AMR

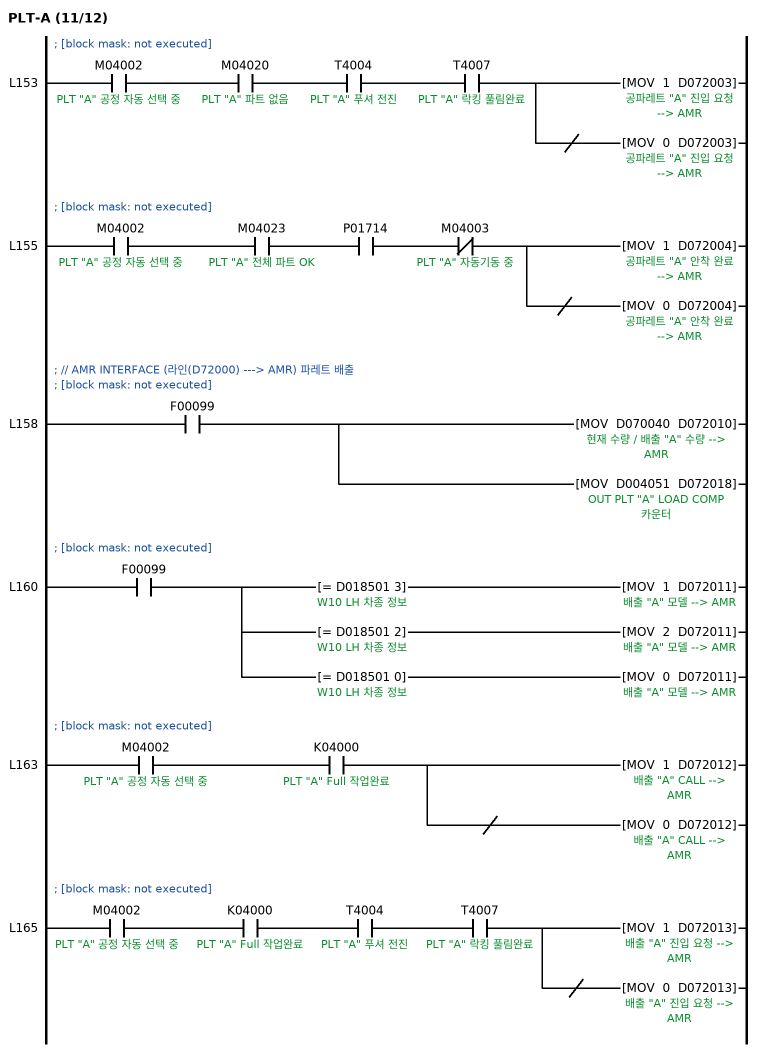
; L153 (block mask: not executed)
LOAD      M04002	// PLT "A" 공정 자동 선택 중
AND       M04020	// PLT "A" 파트 없음
AND       T4004	// PLT "A" 푸셔 전진
AND       T4007	// PLT "A" 락킹 풀림완료
MOV       1 D072003	// 공파레트 "A" 진입 요청 --> AMR
NOT
MOV       0 D072003	// 공파레트 "A" 진입 요청 --> AMR
; L155 (block mask: not executed)
LOAD      M04002	// PLT "A" 공정 자동 선택 중
AND       M04023	// PLT "A" 전체 파트 OK
AND       P01714
AND NOT   M04003	// PLT "A" 자동기동 중
MOV       1 D072004	// 공파레트 "A" 안착 완료 --> AMR
NOT
MOV       0 D072004	// 공파레트 "A" 안착 완료 --> AMR
//   // AMR INTERFACE (라인(D72000) ---> AMR) 파레트 배출
; L158 (block mask: not executed)
LOAD      F00099
MOV       D070040 D072010	// 현재 수량 / 배출 "A" 수량 --> AMR
MOV       D004051 D072018	// OUT PLT "A" LOAD COMP 카운터
; L160 (block mask: not executed)
LOAD      F00099
MPUSH
AND=      D018501 3	// W10 LH 차종 정보
MOV       1 D072011	// 배출 "A" 모델 --> AMR
MLOAD
AND=      D018501 2	// W10 LH 차종 정보
MOV       2 D072011	// 배출 "A" 모델 --> AMR
MPOP
AND=      D018501 0	// W10 LH 차종 정보
MOV       0 D072011	// 배출 "A" 모델 --> AMR
; L163 (block mask: not executed)
LOAD      M04002	// PLT "A" 공정 자동 선택 중
AND       K04000	// PLT "A" Full 작업완료
MOV       1 D072012	// 배출 "A" CALL --> AMR
NOT
MOV       0 D072012	// 배출 "A" CALL --> AMR
; L165 (block mask: not executed)
LOAD      M04002	// PLT "A" 공정 자동 선택 중
AND       K04000	// PLT "A" Full 작업완료
AND       T4004	// PLT "A" 푸셔 전진
AND       T4007	// PLT "A" 락킹 풀림완료
MOV       1 D072013	// 배출 "A" 진입 요청 --> AMR
NOT
MOV       0 D072013	// 배출 "A" 진입 요청 --> AMR

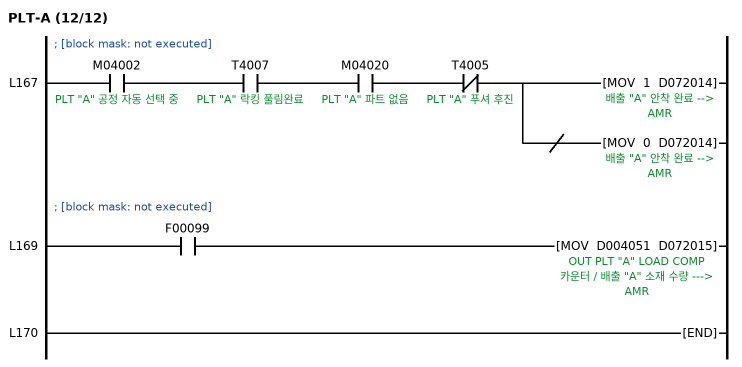
; L167 (block mask: not executed)
LOAD      M04002	// PLT "A" 공정 자동 선택 중
AND       T4007	// PLT "A" 락킹 풀림완료
AND       M04020	// PLT "A" 파트 없음
AND NOT   T4005	// PLT "A" 푸셔 후진
MOV       1 D072014	// 배출 "A" 안착 완료 --> AMR
NOT
MOV       0 D072014	// 배출 "A" 안착 완료 --> AMR
; L169 (block mask: not executed)
LOAD      F00099
MOV       D004051 D072015	// OUT PLT "A" LOAD COMP 카운터 / 배출 "A" 소재 수량 ---> AMR
; L170
END

PROGRAM PLT-B (task: 스캔 프로그램)

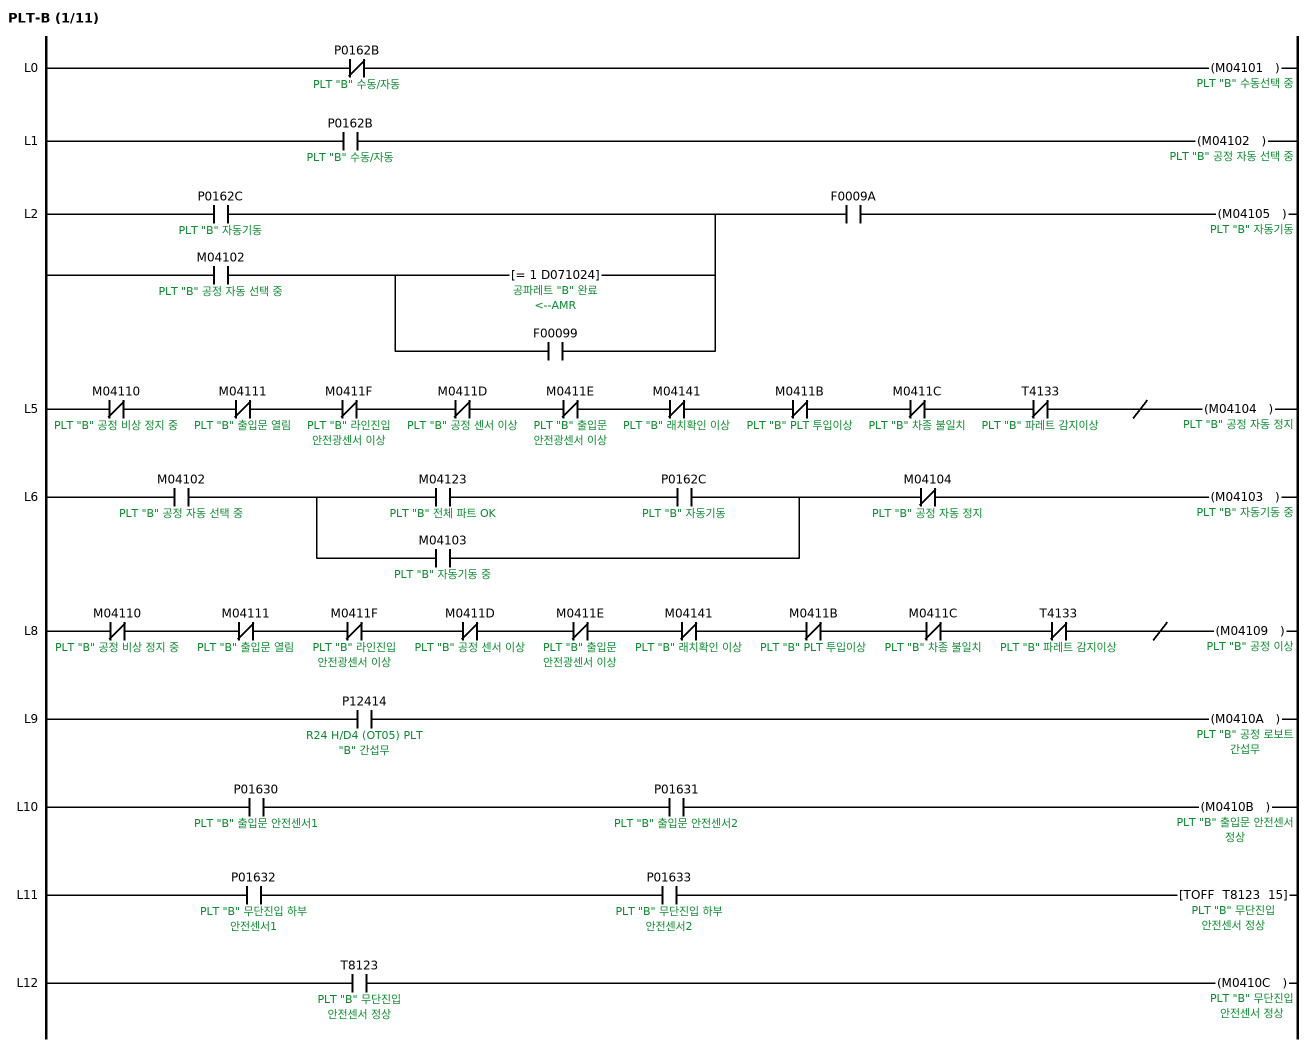
; L0
LOAD NOT  P0162B	// PLT "B" 수동/자동
OUT       M04101	// PLT "B" 수동선택 중
; L1
LOAD      P0162B	// PLT "B" 수동/자동
OUT       M04102	// PLT "B" 공정 자동 선택 중
; L2
LOAD      P0162C	// PLT "B" 자동기동
LOAD      M04102	// PLT "B" 공정 자동 선택 중
LOAD=     1 D071024	// 공파레트 "B" 완료 <--AMR
OR        F00099
AND LOAD
OR LOAD
AND       F0009A
OUT       M04105	// PLT "B" 자동기동
; L5
LOAD NOT  M04110	// PLT "B" 공정 비상 정지 중
AND NOT   M04111	// PLT "B" 출입문 열림
AND NOT   M0411F	// PLT "B" 라인진입 안전광센서 이상
AND NOT   M0411D	// PLT "B" 공정 센서 이상
AND NOT   M0411E	// PLT "B" 출입문 안전광센서 이상
AND NOT   M04141	// PLT "B" 래치확인 이상
AND NOT   M0411B	// PLT "B" PLT 투입이상
AND NOT   M0411C	// PLT "B" 차종 불일치
AND NOT   T4133	// PLT "B" 파레트 감지이상
NOT
OUT       M04104	// PLT "B" 공정 자동 정지
; L6
LOAD      M04102	// PLT "B" 공정 자동 선택 중
LOAD      M04123	// PLT "B" 전체 파트 OK
AND       P0162C	// PLT "B" 자동기동
OR        M04103	// PLT "B" 자동기동 중
AND LOAD
AND NOT   M04104	// PLT "B" 공정 자동 정지
OUT       M04103	// PLT "B" 자동기동 중
; L8
LOAD NOT  M04110	// PLT "B" 공정 비상 정지 중
AND NOT   M04111	// PLT "B" 출입문 열림
AND NOT   M0411F	// PLT "B" 라인진입 안전광센서 이상
AND NOT   M0411D	// PLT "B" 공정 센서 이상
AND NOT   M0411E	// PLT "B" 출입문 안전광센서 이상
AND NOT   M04141	// PLT "B" 래치확인 이상
AND NOT   M0411B	// PLT "B" PLT 투입이상
AND NOT   M0411C	// PLT "B" 차종 불일치
AND NOT   T4133	// PLT "B" 파레트 감지이상
NOT
OUT       M04109	// PLT "B" 공정 이상
; L9
LOAD      P12414	// R24 H/D4 (OT05) PLT "B" 간섭무
OUT       M0410A	// PLT "B" 공정 로보트 간섭무
; L10
LOAD      P01630	// PLT "B" 출입문 안전센서1
AND       P01631	// PLT "B" 출입문 안전센서2
OUT       M0410B	// PLT "B" 출입문 안전센서 정상
; L11
LOAD      P01632	// PLT "B" 무단진입 하부 안전센서1
AND       P01633	// PLT "B" 무단진입 하부 안전센서2
TOFF      T8123 15	// PLT "B" 무단진입 안전센서 정상
; L12
LOAD      T8123	// PLT "B" 무단진입 안전센서 정상
OUT       M0410C	// PLT "B" 무단진입 안전센서 정상

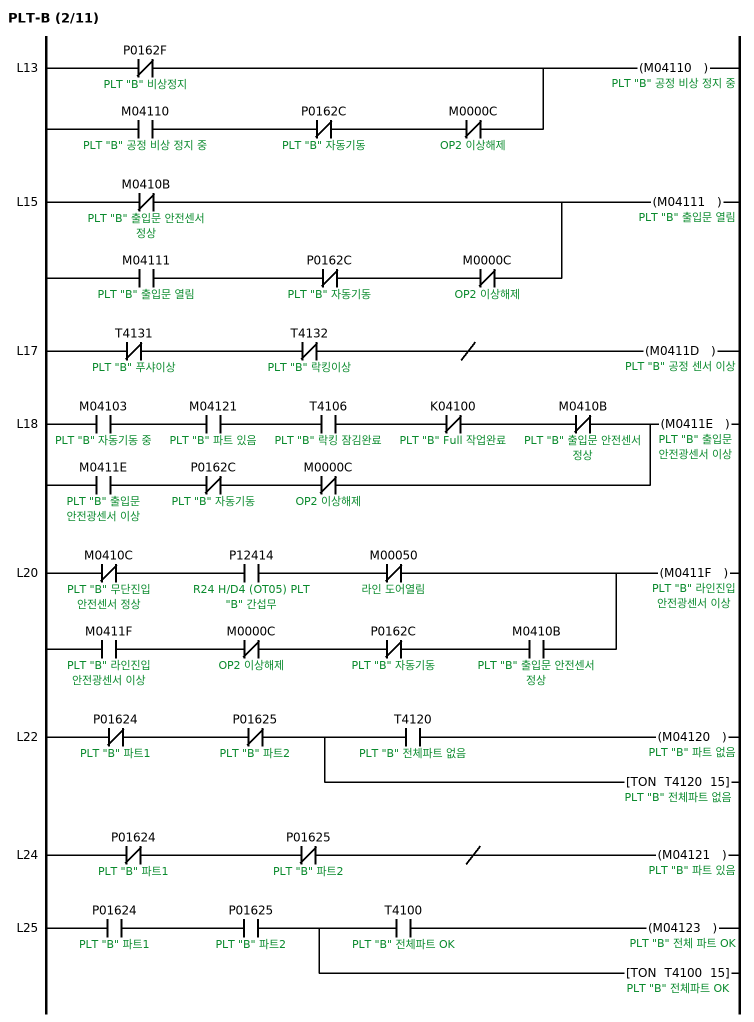
; L13
LOAD NOT  P0162F	// PLT "B" 비상정지
LOAD      M04110	// PLT "B" 공정 비상 정지 중
AND NOT   P0162C	// PLT "B" 자동기동
AND NOT   M0000C	// OP2 이상해제
OR LOAD
OUT       M04110	// PLT "B" 공정 비상 정지 중
; L15
LOAD NOT  M0410B	// PLT "B" 출입문 안전센서 정상
LOAD      M04111	// PLT "B" 출입문 열림
AND NOT   P0162C	// PLT "B" 자동기동
AND NOT   M0000C	// OP2 이상해제
OR LOAD
OUT       M04111	// PLT "B" 출입문 열림
; L17
LOAD NOT  T4131	// PLT "B" 푸샤이상
AND NOT   T4132	// PLT "B" 락킹이상
NOT
OUT       M0411D	// PLT "B" 공정 센서 이상
; L18
LOAD      M04103	// PLT "B" 자동기동 중
AND       M04121	// PLT "B" 파트 있음
AND       T4106	// PLT "B" 락킹 잠김완료
AND NOT   K04100	// PLT "B" Full 작업완료
AND NOT   M0410B	// PLT "B" 출입문 안전센서 정상
LOAD      M0411E	// PLT "B" 출입문 안전광센서 이상
AND NOT   P0162C	// PLT "B" 자동기동
AND NOT   M0000C	// OP2 이상해제
OR LOAD
OUT       M0411E	// PLT "B" 출입문 안전광센서 이상
; L20
LOAD NOT  M0410C	// PLT "B" 무단진입 안전센서 정상
AND       P12414	// R24 H/D4 (OT05) PLT "B" 간섭무
AND NOT   M00050	// 라인 도어열림
LOAD      M0411F	// PLT "B" 라인진입 안전광센서 이상
AND NOT   M0000C	// OP2 이상해제
AND NOT   P0162C	// PLT "B" 자동기동
AND       M0410B	// PLT "B" 출입문 안전센서 정상
OR LOAD
OUT       M0411F	// PLT "B" 라인진입 안전광센서 이상
; L22
LOAD NOT  P01624	// PLT "B" 파트1
AND NOT   P01625	// PLT "B" 파트2
MPUSH
AND       T4120	// PLT "B" 전체파트 없음
OUT       M04120	// PLT "B" 파트 없음
MPOP
TON       T4120 15	// PLT "B" 전체파트 없음
; L24
LOAD NOT  P01624	// PLT "B" 파트1
AND NOT   P01625	// PLT "B" 파트2
NOT
OUT       M04121	// PLT "B" 파트 있음
; L25
LOAD      P01624	// PLT "B" 파트1
AND       P01625	// PLT "B" 파트2
MPUSH
AND       T4100	// PLT "B" 전체파트 OK
OUT       M04123	// PLT "B" 전체 파트 OK
MPOP
TON       T4100 15	// PLT "B" 전체파트 OK

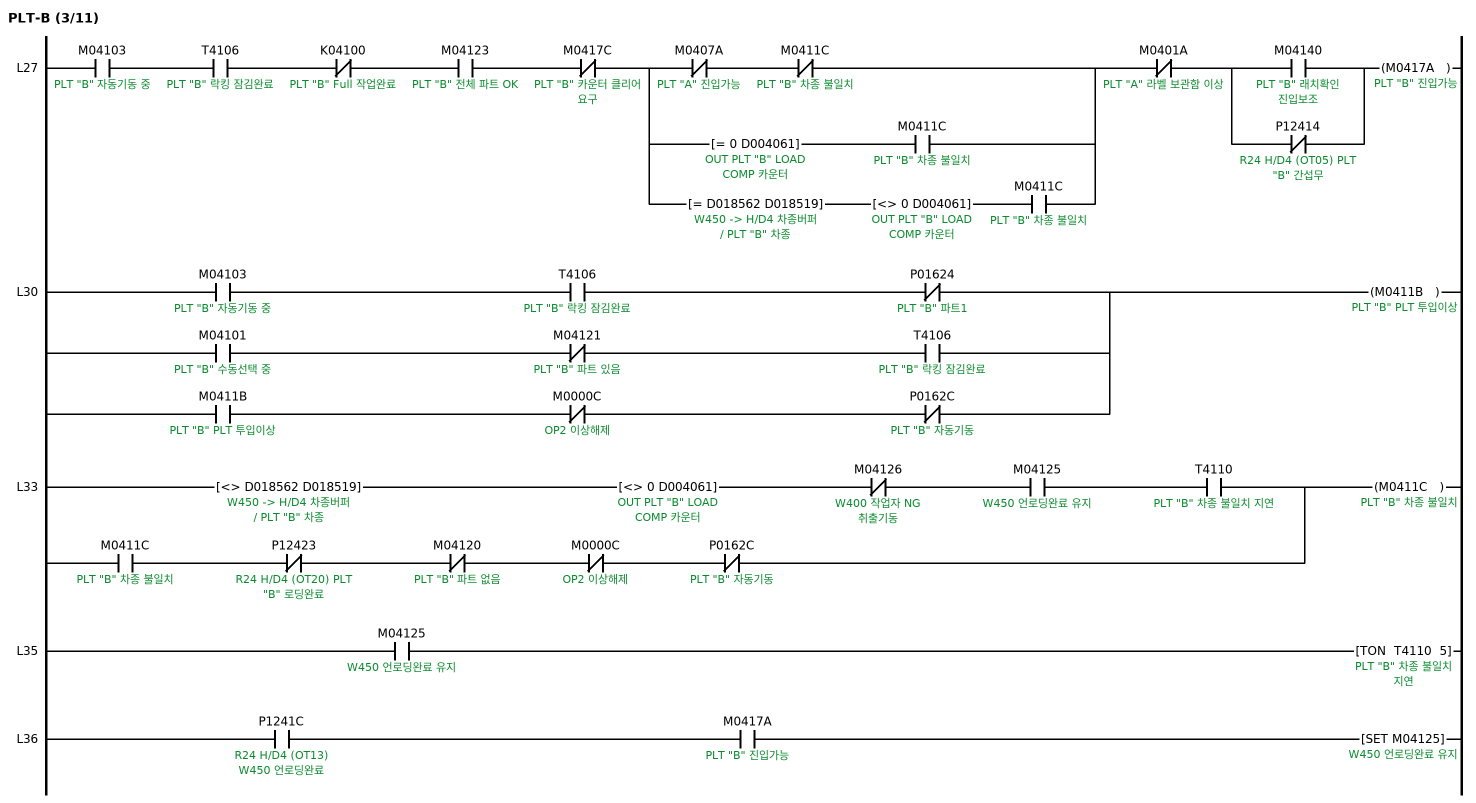
; L27
LOAD      M04103	// PLT "B" 자동기동 중
AND       T4106	// PLT "B" 락킹 잠김완료
AND NOT   K04100	// PLT "B" Full 작업완료
AND       M04123	// PLT "B" 전체 파트 OK
AND NOT   M0417C	// PLT "B" 카운터 클리어 요구
LOAD NOT  M0407A	// PLT "A" 진입가능
AND NOT   M0411C	// PLT "B" 차종 불일치
LOAD=     0 D004061	// OUT PLT "B" LOAD COMP 카운터
AND       M0411C	// PLT "B" 차종 불일치
OR LOAD
LOAD=     D018562 D018519	// W450 -> H/D4 차종버퍼 / PLT "B" 차종
AND<>     0 D004061	// OUT PLT "B" LOAD COMP 카운터
AND       M0411C	// PLT "B" 차종 불일치
OR LOAD
AND LOAD
AND NOT   M0401A	// PLT "A" 라벨 보관함 이상
LOAD      M04140	// PLT "B" 래치확인 진입보조
OR NOT    P12414	// R24 H/D4 (OT05) PLT "B" 간섭무
AND LOAD
OUT       M0417A	// PLT "B" 진입가능
; L30
LOAD      M04103	// PLT "B" 자동기동 중
AND       T4106	// PLT "B" 락킹 잠김완료
AND NOT   P01624	// PLT "B" 파트1
LOAD      M04101	// PLT "B" 수동선택 중
AND NOT   M04121	// PLT "B" 파트 있음
AND       T4106	// PLT "B" 락킹 잠김완료
OR LOAD
LOAD      M0411B	// PLT "B" PLT 투입이상
AND NOT   M0000C	// OP2 이상해제
AND NOT   P0162C	// PLT "B" 자동기동
OR LOAD
OUT       M0411B	// PLT "B" PLT 투입이상
; L33
LOAD<>    D018562 D018519	// W450 -> H/D4 차종버퍼 / PLT "B" 차종
AND<>     0 D004061	// OUT PLT "B" LOAD COMP 카운터
AND NOT   M04126	// W400 작업자 NG 취출기동
AND       M04125	// W450 언로딩완료 유지
AND       T4110	// PLT "B" 차종 불일치 지연
LOAD      M0411C	// PLT "B" 차종 불일치
AND NOT   P12423	// R24 H/D4 (OT20) PLT "B" 로딩완료
AND NOT   M04120	// PLT "B" 파트 없음
AND NOT   M0000C	// OP2 이상해제
AND NOT   P0162C	// PLT "B" 자동기동
OR LOAD
OUT       M0411C	// PLT "B" 차종 불일치
; L35
LOAD      M04125	// W450 언로딩완료 유지
TON       T4110 5	// PLT "B" 차종 불일치 지연
; L36
LOAD      P1241C	// R24 H/D4 (OT13) W450 언로딩완료
AND       M0417A	// PLT "B" 진입가능
SET       M04125	// W450 언로딩완료 유지

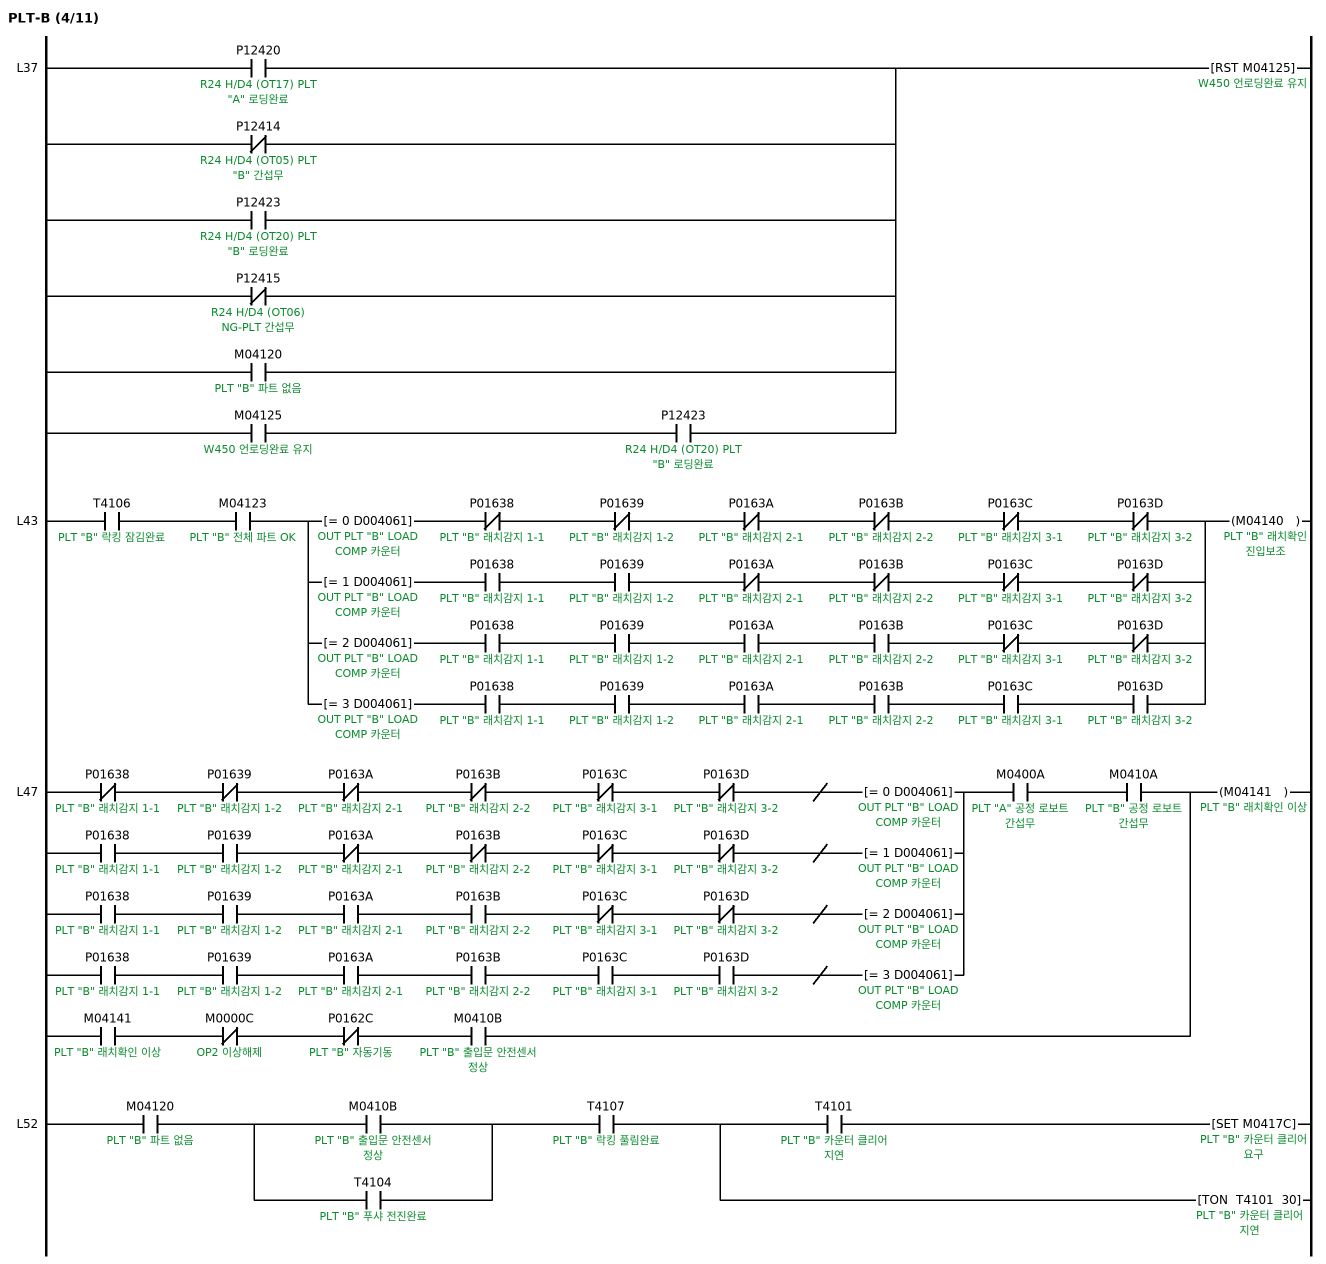
; L37
LOAD      P12420	// R24 H/D4 (OT17) PLT "A" 로딩완료
OR NOT    P12414	// R24 H/D4 (OT05) PLT "B" 간섭무
OR        P12423	// R24 H/D4 (OT20) PLT "B" 로딩완료
OR NOT    P12415	// R24 H/D4 (OT06) NG-PLT 간섭무
OR        M04120	// PLT "B" 파트 없음
LOAD      M04125	// W450 언로딩완료 유지
AND       P12423	// R24 H/D4 (OT20) PLT "B" 로딩완료
OR LOAD
RST       M04125	// W450 언로딩완료 유지
; L43
LOAD      T4106	// PLT "B" 락킹 잠김완료
AND       M04123	// PLT "B" 전체 파트 OK
LOAD=     0 D004061	// OUT PLT "B" LOAD COMP 카운터
AND NOT   P01638	// PLT "B" 래치감지 1-1
AND NOT   P01639	// PLT "B" 래치감지 1-2
AND NOT   P0163A	// PLT "B" 래치감지 2-1
AND NOT   P0163B	// PLT "B" 래치감지 2-2
AND NOT   P0163C	// PLT "B" 래치감지 3-1
AND NOT   P0163D	// PLT "B" 래치감지 3-2
LOAD=     1 D004061	// OUT PLT "B" LOAD COMP 카운터
AND       P01638	// PLT "B" 래치감지 1-1
AND       P01639	// PLT "B" 래치감지 1-2
AND NOT   P0163A	// PLT "B" 래치감지 2-1
AND NOT   P0163B	// PLT "B" 래치감지 2-2
AND NOT   P0163C	// PLT "B" 래치감지 3-1
AND NOT   P0163D	// PLT "B" 래치감지 3-2
OR LOAD
LOAD=     2 D004061	// OUT PLT "B" LOAD COMP 카운터
AND       P01638	// PLT "B" 래치감지 1-1
AND       P01639	// PLT "B" 래치감지 1-2
AND       P0163A	// PLT "B" 래치감지 2-1
AND       P0163B	// PLT "B" 래치감지 2-2
AND NOT   P0163C	// PLT "B" 래치감지 3-1
AND NOT   P0163D	// PLT "B" 래치감지 3-2
OR LOAD
LOAD=     3 D004061	// OUT PLT "B" LOAD COMP 카운터
AND       P01638	// PLT "B" 래치감지 1-1
AND       P01639	// PLT "B" 래치감지 1-2
AND       P0163A	// PLT "B" 래치감지 2-1
AND       P0163B	// PLT "B" 래치감지 2-2
AND       P0163C	// PLT "B" 래치감지 3-1
AND       P0163D	// PLT "B" 래치감지 3-2
OR LOAD
AND LOAD
OUT       M04140	// PLT "B" 래치확인 진입보조
; L47
LOAD NOT  P01638	// PLT "B" 래치감지 1-1
AND NOT   P01639	// PLT "B" 래치감지 1-2
AND NOT   P0163A	// PLT "B" 래치감지 2-1
AND NOT   P0163B	// PLT "B" 래치감지 2-2
AND NOT   P0163C	// PLT "B" 래치감지 3-1
AND NOT   P0163D	// PLT "B" 래치감지 3-2
NOT
AND=      0 D004061	// OUT PLT "B" LOAD COMP 카운터
LOAD      P01638	// PLT "B" 래치감지 1-1
AND       P01639	// PLT "B" 래치감지 1-2
AND NOT   P0163A	// PLT "B" 래치감지 2-1
AND NOT   P0163B	// PLT "B" 래치감지 2-2
AND NOT   P0163C	// PLT "B" 래치감지 3-1
AND NOT   P0163D	// PLT "B" 래치감지 3-2
NOT
AND=      1 D004061	// OUT PLT "B" LOAD COMP 카운터
OR LOAD
LOAD      P01638	// PLT "B" 래치감지 1-1
AND       P01639	// PLT "B" 래치감지 1-2
AND       P0163A	// PLT "B" 래치감지 2-1
AND       P0163B	// PLT "B" 래치감지 2-2
AND NOT   P0163C	// PLT "B" 래치감지 3-1
AND NOT   P0163D	// PLT "B" 래치감지 3-2
NOT
AND=      2 D004061	// OUT PLT "B" LOAD COMP 카운터
OR LOAD
LOAD      P01638	// PLT "B" 래치감지 1-1
AND       P01639	// PLT "B" 래치감지 1-2
AND       P0163A	// PLT "B" 래치감지 2-1
AND       P0163B	// PLT "B" 래치감지 2-2
AND       P0163C	// PLT "B" 래치감지 3-1
AND       P0163D	// PLT "B" 래치감지 3-2
NOT
AND=      3 D004061	// OUT PLT "B" LOAD COMP 카운터
OR LOAD
AND       M0400A	// PLT "A" 공정 로보트 간섭무
AND       M0410A	// PLT "B" 공정 로보트 간섭무
LOAD      M04141	// PLT "B" 래치확인 이상
AND NOT   M0000C	// OP2 이상해제
AND NOT   P0162C	// PLT "B" 자동기동
AND       M0410B	// PLT "B" 출입문 안전센서 정상
OR LOAD
OUT       M04141	// PLT "B" 래치확인 이상
; L52
LOAD      M04120	// PLT "B" 파트 없음
LOAD      M0410B	// PLT "B" 출입문 안전센서 정상
OR        T4104	// PLT "B" 푸샤 전진완료
AND LOAD
AND       T4107	// PLT "B" 락킹 풀림완료
MPUSH
AND       T4101	// PLT "B" 카운터 클리어 지연
SET       M0417C	// PLT "B" 카운터 클리어 요구
MPOP
TON       T4101 30	// PLT "B" 카운터 클리어 지연

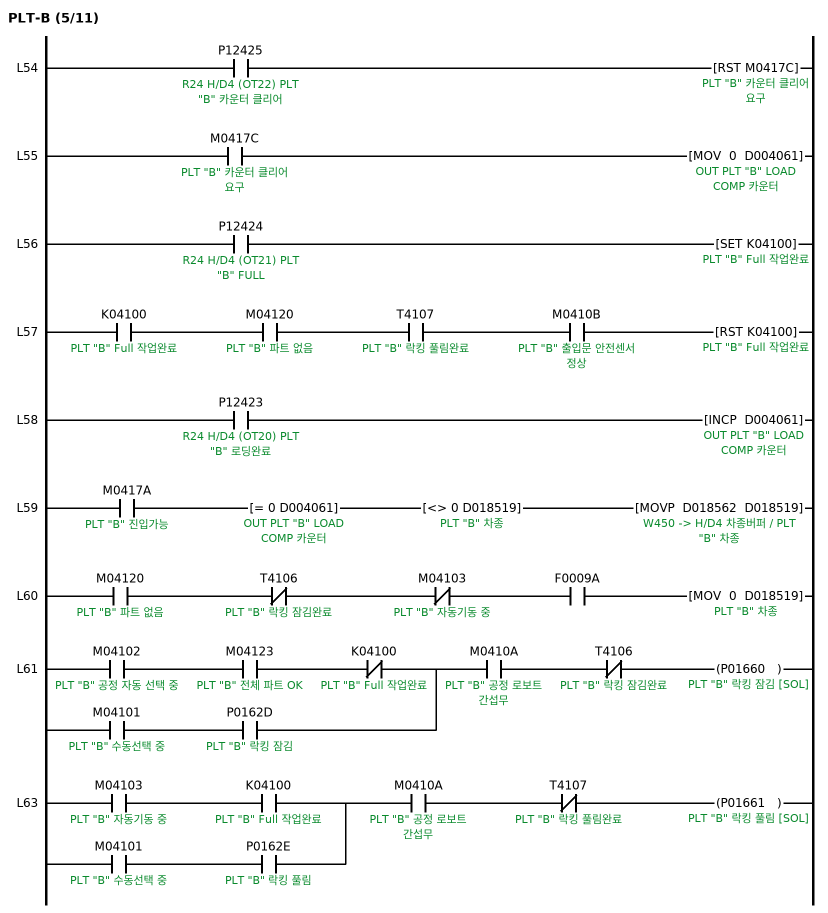
; L54
LOAD      P12425	// R24 H/D4 (OT22) PLT "B" 카운터 클리어
RST       M0417C	// PLT "B" 카운터 클리어 요구
; L55
LOAD      M0417C	// PLT "B" 카운터 클리어 요구
MOV       0 D004061	// OUT PLT "B" LOAD COMP 카운터
; L56
LOAD      P12424	// R24 H/D4 (OT21) PLT "B" FULL
SET       K04100	// PLT "B" Full 작업완료
; L57
LOAD      K04100	// PLT "B" Full 작업완료
AND       M04120	// PLT "B" 파트 없음
AND       T4107	// PLT "B" 락킹 풀림완료
AND       M0410B	// PLT "B" 출입문 안전센서 정상
RST       K04100	// PLT "B" Full 작업완료
; L58
LOAD      P12423	// R24 H/D4 (OT20) PLT "B" 로딩완료
INCP      D004061	// OUT PLT "B" LOAD COMP 카운터
; L59
LOAD      M0417A	// PLT "B" 진입가능
AND=      0 D004061	// OUT PLT "B" LOAD COMP 카운터
AND<>     0 D018519	// PLT "B" 차종
MOVP      D018562 D018519	// W450 -> H/D4 차종버퍼 / PLT "B" 차종
; L60
LOAD      M04120	// PLT "B" 파트 없음
AND NOT   T4106	// PLT "B" 락킹 잠김완료
AND NOT   M04103	// PLT "B" 자동기동 중
AND       F0009A
MOV       0 D018519	// PLT "B" 차종
; L61
LOAD      M04102	// PLT "B" 공정 자동 선택 중
AND       M04123	// PLT "B" 전체 파트 OK
AND NOT   K04100	// PLT "B" Full 작업완료
LOAD      M04101	// PLT "B" 수동선택 중
AND       P0162D	// PLT "B" 락킹 잠김
OR LOAD
AND       M0410A	// PLT "B" 공정 로보트 간섭무
AND NOT   T4106	// PLT "B" 락킹 잠김완료
OUT       P01660	// PLT "B" 락킹 잠김 [SOL]
; L63
LOAD      M04103	// PLT "B" 자동기동 중
AND       K04100	// PLT "B" Full 작업완료
LOAD      M04101	// PLT "B" 수동선택 중
AND       P0162E	// PLT "B" 락킹 풀림
OR LOAD
AND       M0410A	// PLT "B" 공정 로보트 간섭무
AND NOT   T4107	// PLT "B" 락킹 풀림완료
OUT       P01661	// PLT "B" 락킹 풀림 [SOL]

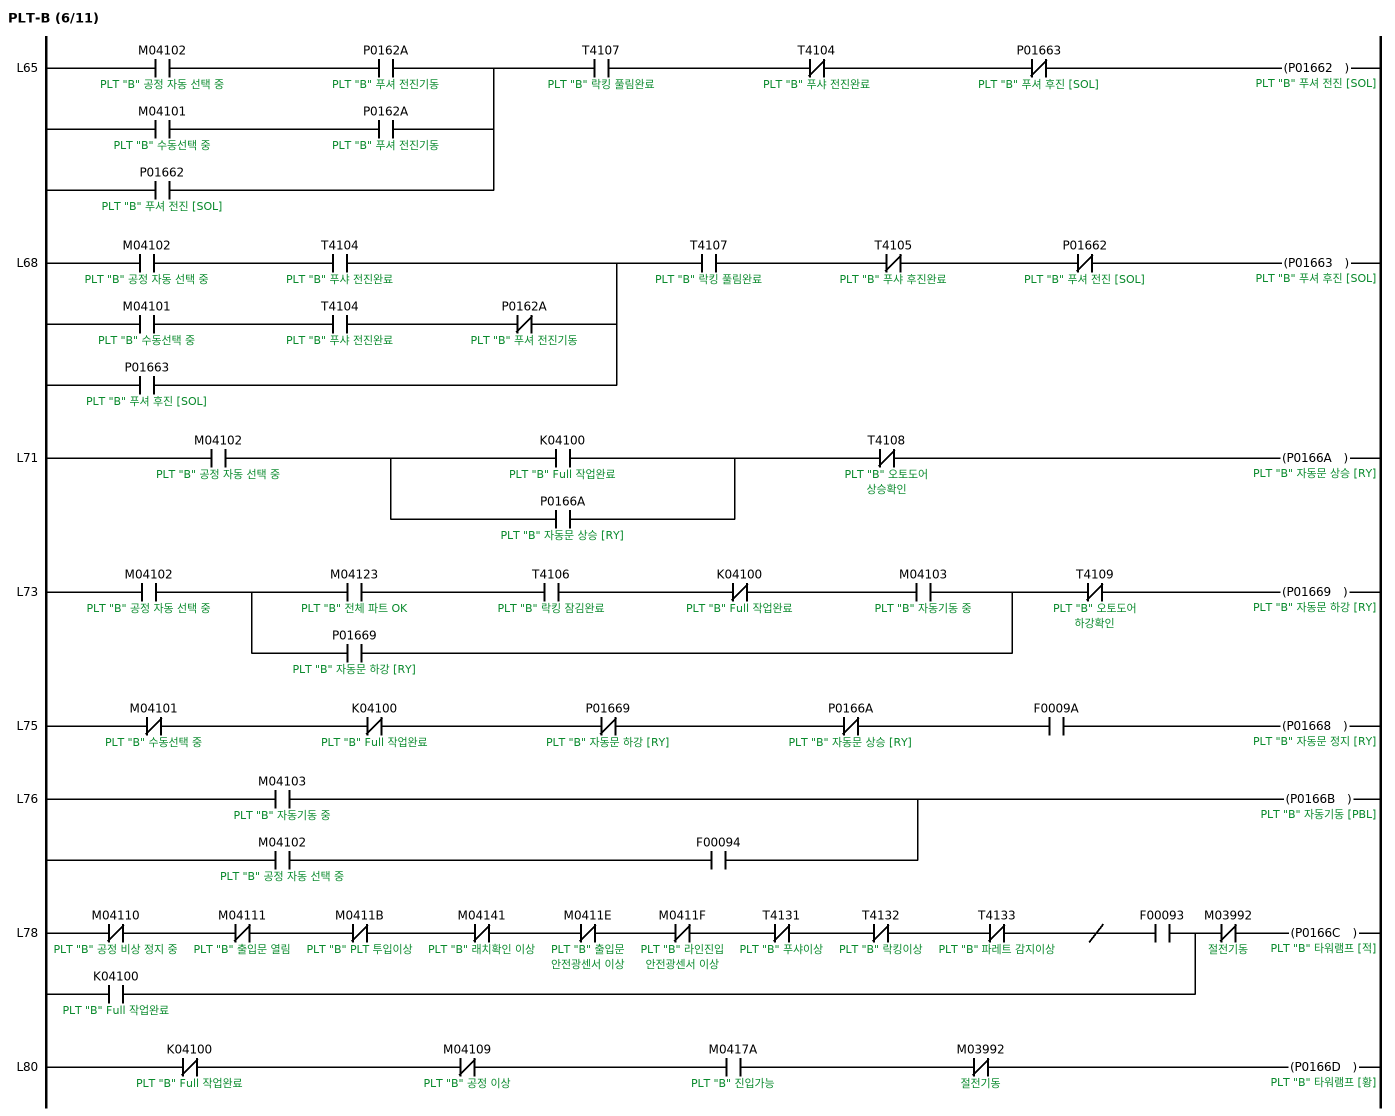
; L65
LOAD      M04102	// PLT "B" 공정 자동 선택 중
AND       P0162A	// PLT "B" 푸셔 전진기동
LOAD      M04101	// PLT "B" 수동선택 중
AND       P0162A	// PLT "B" 푸셔 전진기동
OR LOAD
OR        P01662	// PLT "B" 푸셔 전진 [SOL]
AND       T4107	// PLT "B" 락킹 풀림완료
AND NOT   T4104	// PLT "B" 푸샤 전진완료
AND NOT   P01663	// PLT "B" 푸셔 후진 [SOL]
OUT       P01662	// PLT "B" 푸셔 전진 [SOL]
; L68
LOAD      M04102	// PLT "B" 공정 자동 선택 중
AND       T4104	// PLT "B" 푸샤 전진완료
LOAD      M04101	// PLT "B" 수동선택 중
AND       T4104	// PLT "B" 푸샤 전진완료
AND NOT   P0162A	// PLT "B" 푸셔 전진기동
OR LOAD
OR        P01663	// PLT "B" 푸셔 후진 [SOL]
AND       T4107	// PLT "B" 락킹 풀림완료
AND NOT   T4105	// PLT "B" 푸샤 후진완료
AND NOT   P01662	// PLT "B" 푸셔 전진 [SOL]
OUT       P01663	// PLT "B" 푸셔 후진 [SOL]
; L71
LOAD      M04102	// PLT "B" 공정 자동 선택 중
LOAD      K04100	// PLT "B" Full 작업완료
OR        P0166A	// PLT "B" 자동문 상승 [RY]
AND LOAD
AND NOT   T4108	// PLT "B" 오토도어 상승확인
OUT       P0166A	// PLT "B" 자동문 상승 [RY]
; L73
LOAD      M04102	// PLT "B" 공정 자동 선택 중
LOAD      M04123	// PLT "B" 전체 파트 OK
AND       T4106	// PLT "B" 락킹 잠김완료
AND NOT   K04100	// PLT "B" Full 작업완료
AND       M04103	// PLT "B" 자동기동 중
OR        P01669	// PLT "B" 자동문 하강 [RY]
AND LOAD
AND NOT   T4109	// PLT "B" 오토도어 하강확인
OUT       P01669	// PLT "B" 자동문 하강 [RY]
; L75
LOAD NOT  M04101	// PLT "B" 수동선택 중
AND NOT   K04100	// PLT "B" Full 작업완료
AND NOT   P01669	// PLT "B" 자동문 하강 [RY]
AND NOT   P0166A	// PLT "B" 자동문 상승 [RY]
AND       F0009A
OUT       P01668	// PLT "B" 자동문 정지 [RY]
; L76
LOAD      M04103	// PLT "B" 자동기동 중
LOAD      M04102	// PLT "B" 공정 자동 선택 중
AND       F00094
OR LOAD
OUT       P0166B	// PLT "B" 자동기동 [PBL]
; L78
LOAD NOT  M04110	// PLT "B" 공정 비상 정지 중
AND NOT   M04111	// PLT "B" 출입문 열림
AND NOT   M0411B	// PLT "B" PLT 투입이상
AND NOT   M04141	// PLT "B" 래치확인 이상
AND NOT   M0411E	// PLT "B" 출입문 안전광센서 이상
AND NOT   M0411F	// PLT "B" 라인진입 안전광센서 이상
AND NOT   T4131	// PLT "B" 푸샤이상
AND NOT   T4132	// PLT "B" 락킹이상
AND NOT   T4133	// PLT "B" 파레트 감지이상
NOT
AND       F00093
OR        K04100	// PLT "B" Full 작업완료
AND NOT   M03992	// 절전기동
OUT       P0166C	// PLT "B" 타워램프 [적]
; L80
LOAD NOT  K04100	// PLT "B" Full 작업완료
AND NOT   M04109	// PLT "B" 공정 이상
AND       M0417A	// PLT "B" 진입가능
AND NOT   M03992	// 절전기동
OUT       P0166D	// PLT "B" 타워램프 [황]

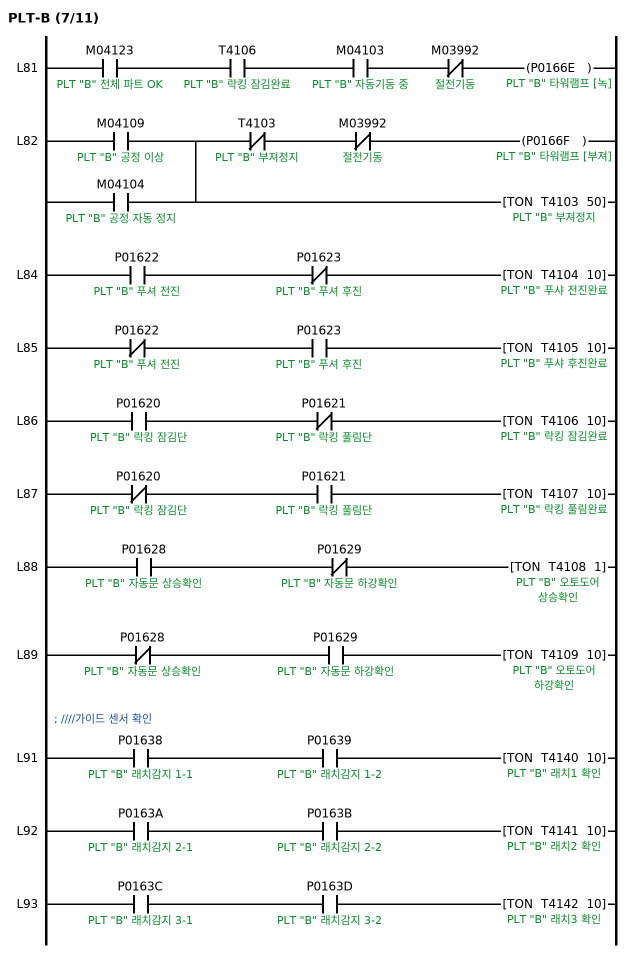
; L81
LOAD      M04123	// PLT "B" 전체 파트 OK
AND       T4106	// PLT "B" 락킹 잠김완료
AND       M04103	// PLT "B" 자동기동 중
AND NOT   M03992	// 절전기동
OUT       P0166E	// PLT "B" 타워램프 [녹]
; L82
LOAD      M04109	// PLT "B" 공정 이상
OR        M04104	// PLT "B" 공정 자동 정지
MPUSH
AND NOT   T4103	// PLT "B" 부져정지
AND NOT   M03992	// 절전기동
OUT       P0166F	// PLT "B" 타워램프 [부져]
MPOP
TON       T4103 50	// PLT "B" 부져정지
; L84
LOAD      P01622	// PLT "B" 푸셔 전진
AND NOT   P01623	// PLT "B" 푸셔 후진
TON       T4104 10	// PLT "B" 푸샤 전진완료
; L85
LOAD NOT  P01622	// PLT "B" 푸셔 전진
AND       P01623	// PLT "B" 푸셔 후진
TON       T4105 10	// PLT "B" 푸샤 후진완료
; L86
LOAD      P01620	// PLT "B" 락킹 잠김단
AND NOT   P01621	// PLT "B" 락킹 풀림단
TON       T4106 10	// PLT "B" 락킹 잠김완료
; L87
LOAD NOT  P01620	// PLT "B" 락킹 잠김단
AND       P01621	// PLT "B" 락킹 풀림단
TON       T4107 10	// PLT "B" 락킹 풀림완료
; L88
LOAD      P01628	// PLT "B" 자동문 상승확인
AND NOT   P01629	// PLT "B" 자동문 하강확인
TON       T4108 1	// PLT "B" 오토도어 상승확인
; L89
LOAD NOT  P01628	// PLT "B" 자동문 상승확인
AND       P01629	// PLT "B" 자동문 하강확인
TON       T4109 10	// PLT "B" 오토도어 하강확인
// ////가이드 센서 확인
; L91
LOAD      P01638	// PLT "B" 래치감지 1-1
AND       P01639	// PLT "B" 래치감지 1-2
TON       T4140 10	// PLT "B" 래치1 확인
; L92
LOAD      P0163A	// PLT "B" 래치감지 2-1
AND       P0163B	// PLT "B" 래치감지 2-2
TON       T4141 10	// PLT "B" 래치2 확인
; L93
LOAD      P0163C	// PLT "B" 래치감지 3-1
AND       P0163D	// PLT "B" 래치감지 3-2
TON       T4142 10	// PLT "B" 래치3 확인

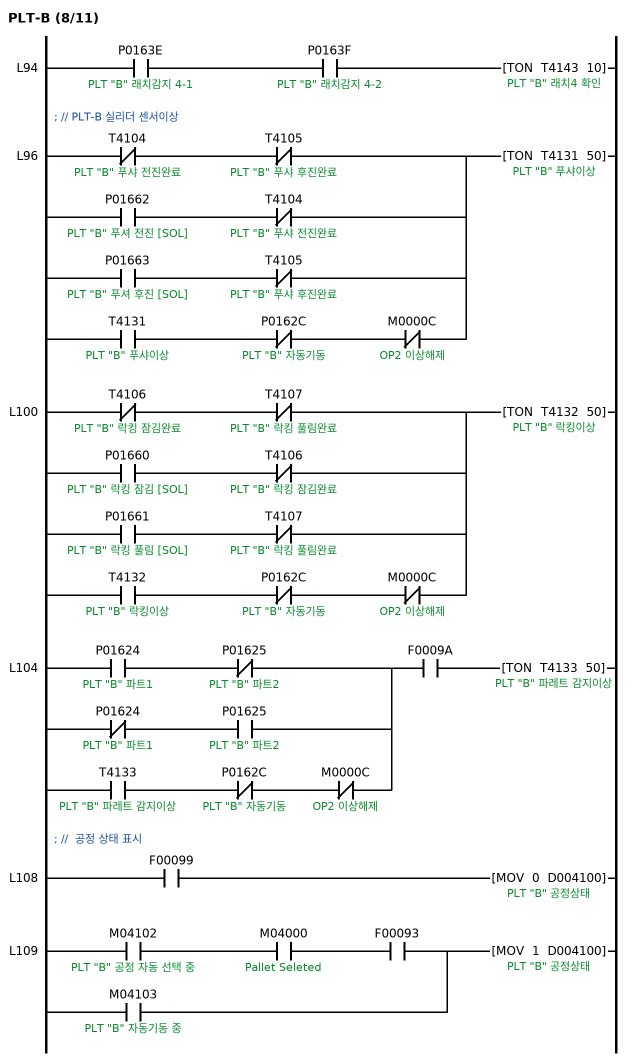
; L94
LOAD      P0163E	// PLT "B" 래치감지 4-1
AND       P0163F	// PLT "B" 래치감지 4-2
TON       T4143 10	// PLT "B" 래치4 확인
// // PLT-B 실리더 센서이상
; L96
LOAD NOT  T4104	// PLT "B" 푸샤 전진완료
AND NOT   T4105	// PLT "B" 푸샤 후진완료
LOAD      P01662	// PLT "B" 푸셔 전진 [SOL]
AND NOT   T4104	// PLT "B" 푸샤 전진완료
OR LOAD
LOAD      P01663	// PLT "B" 푸셔 후진 [SOL]
AND NOT   T4105	// PLT "B" 푸샤 후진완료
OR LOAD
LOAD      T4131	// PLT "B" 푸샤이상
AND NOT   P0162C	// PLT "B" 자동기동
AND NOT   M0000C	// OP2 이상해제
OR LOAD
TON       T4131 50	// PLT "B" 푸샤이상
; L100
LOAD NOT  T4106	// PLT "B" 락킹 잠김완료
AND NOT   T4107	// PLT "B" 락킹 풀림완료
LOAD      P01660	// PLT "B" 락킹 잠김 [SOL]
AND NOT   T4106	// PLT "B" 락킹 잠김완료
OR LOAD
LOAD      P01661	// PLT "B" 락킹 풀림 [SOL]
AND NOT   T4107	// PLT "B" 락킹 풀림완료
OR LOAD
LOAD      T4132	// PLT "B" 락킹이상
AND NOT   P0162C	// PLT "B" 자동기동
AND NOT   M0000C	// OP2 이상해제
OR LOAD
TON       T4132 50	// PLT "B" 락킹이상
; L104
LOAD      P01624	// PLT "B" 파트1
AND NOT   P01625	// PLT "B" 파트2
LOAD NOT  P01624	// PLT "B" 파트1
AND       P01625	// PLT "B" 파트2
OR LOAD
LOAD      T4133	// PLT "B" 파레트 감지이상
AND NOT   P0162C	// PLT "B" 자동기동
AND NOT   M0000C	// OP2 이상해제
OR LOAD
AND       F0009A
TON       T4133 50	// PLT "B" 파레트 감지이상
//   //  공정 상태 표시
; L108
LOAD      F00099
MOV       0 D004100	// PLT "B" 공정상태
; L109
LOAD      M04102	// PLT "B" 공정 자동 선택 중
AND       M04000	// Pallet Seleted
AND       F00093
OR        M04103	// PLT "B" 자동기동 중
MOV       1 D004100	// PLT "B" 공정상태

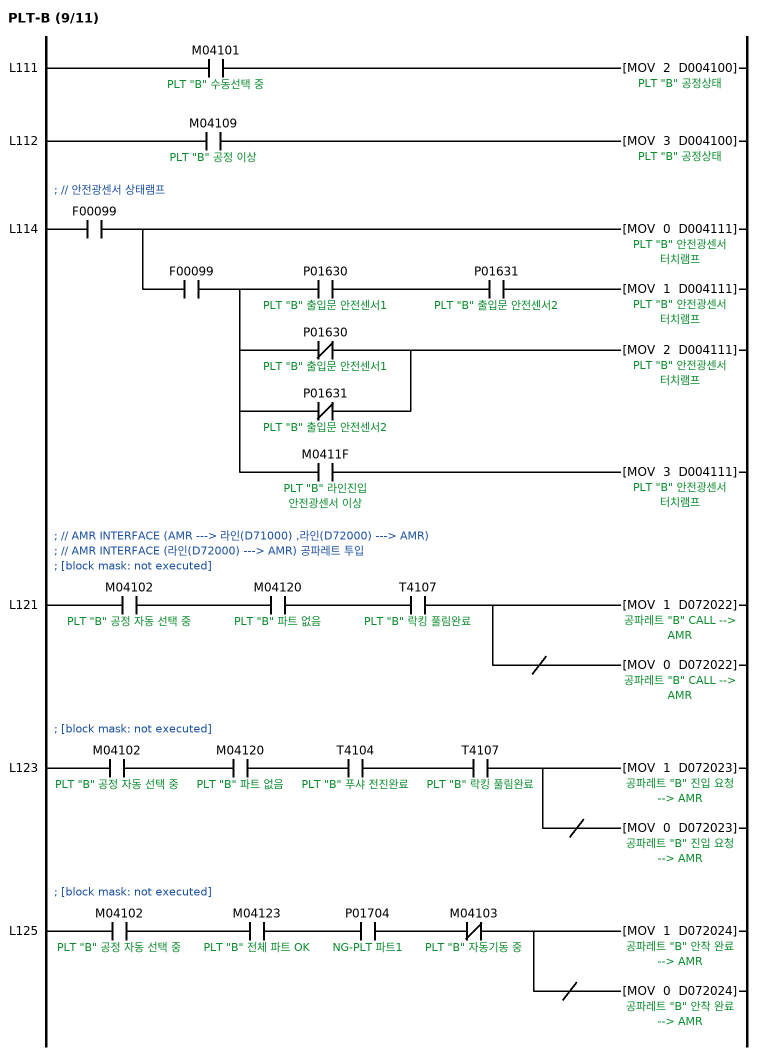
; L111
LOAD      M04101	// PLT "B" 수동선택 중
MOV       2 D004100	// PLT "B" 공정상태
; L112
LOAD      M04109	// PLT "B" 공정 이상
MOV       3 D004100	// PLT "B" 공정상태
//   // 안전광센서 상태램프
; L114
LOAD      F00099
MOV       0 D004111	// PLT "B" 안전광센서 터치램프
AND       F00099
MPUSH
AND       P01630	// PLT "B" 출입문 안전센서1
AND       P01631	// PLT "B" 출입문 안전센서2
MOV       1 D004111	// PLT "B" 안전광센서 터치램프
MLOAD
LOAD NOT  P01630	// PLT "B" 출입문 안전센서1
OR NOT    P01631	// PLT "B" 출입문 안전센서2
AND LOAD
MOV       2 D004111	// PLT "B" 안전광센서 터치램프
MPOP
AND       M0411F	// PLT "B" 라인진입 안전광센서 이상
MOV       3 D004111	// PLT "B" 안전광센서 터치램프
//   // AMR INTERFACE (AMR ---> 라인(D71000) ,라인(D72000) ---> AMR)
//   // AMR INTERFACE (라인(D72000) ---> AMR) 공파레트 투입
; L121 (block mask: not executed)
LOAD      M04102	// PLT "B" 공정 자동 선택 중
AND       M04120	// PLT "B" 파트 없음
AND       T4107	// PLT "B" 락킹 풀림완료
MOV       1 D072022	// 공파레트 "B" CALL --> AMR
NOT
MOV       0 D072022	// 공파레트 "B" CALL --> AMR
; L123 (block mask: not executed)
LOAD      M04102	// PLT "B" 공정 자동 선택 중
AND       M04120	// PLT "B" 파트 없음
AND       T4104	// PLT "B" 푸샤 전진완료
AND       T4107	// PLT "B" 락킹 풀림완료
MOV       1 D072023	// 공파레트 "B" 진입 요청 --> AMR
NOT
MOV       0 D072023	// 공파레트 "B" 진입 요청 --> AMR
; L125 (block mask: not executed)
LOAD      M04102	// PLT "B" 공정 자동 선택 중
AND       M04123	// PLT "B" 전체 파트 OK
AND       P01704	// NG-PLT 파트1
AND NOT   M04103	// PLT "B" 자동기동 중
MOV       1 D072024	// 공파레트 "B" 안착 완료 --> AMR
NOT
MOV       0 D072024	// 공파레트 "B" 안착 완료 --> AMR

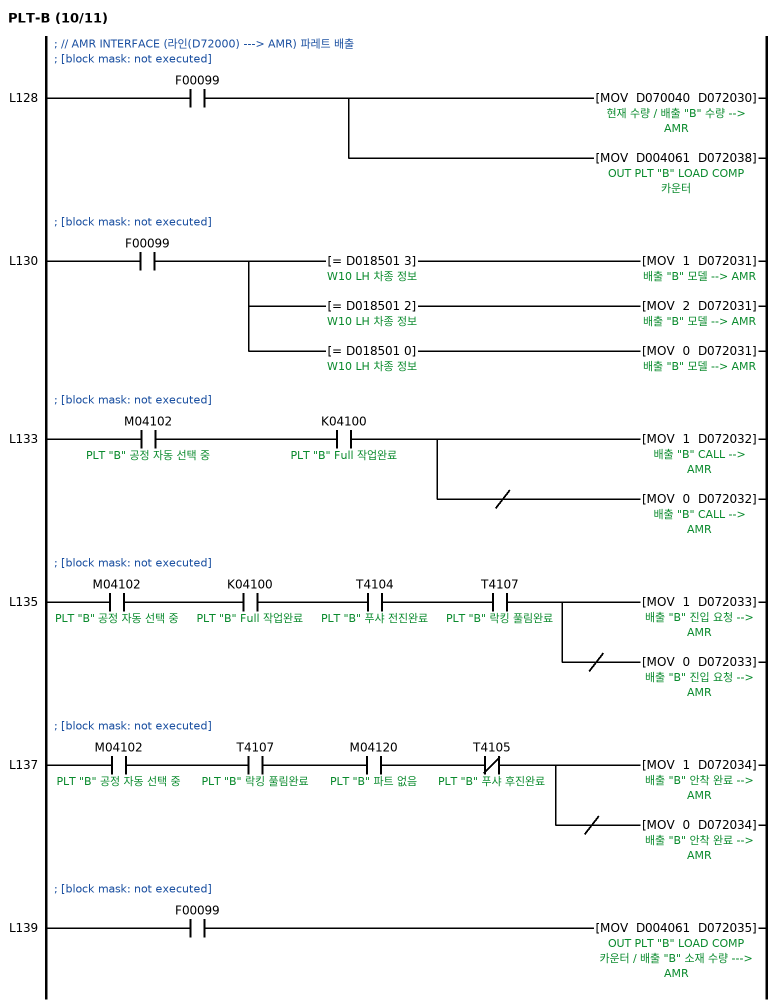
//   // AMR INTERFACE (라인(D72000) ---> AMR) 파레트 배출
; L128 (block mask: not executed)
LOAD      F00099
MOV       D070040 D072030	// 현재 수량 / 배출 "B" 수량 --> AMR
MOV       D004061 D072038	// OUT PLT "B" LOAD COMP 카운터
; L130 (block mask: not executed)
LOAD      F00099
MPUSH
AND=      D018501 3	// W10 LH 차종 정보
MOV       1 D072031	// 배출 "B" 모델 --> AMR
MLOAD
AND=      D018501 2	// W10 LH 차종 정보
MOV       2 D072031	// 배출 "B" 모델 --> AMR
MPOP
AND=      D018501 0	// W10 LH 차종 정보
MOV       0 D072031	// 배출 "B" 모델 --> AMR
; L133 (block mask: not executed)
LOAD      M04102	// PLT "B" 공정 자동 선택 중
AND       K04100	// PLT "B" Full 작업완료
MOV       1 D072032	// 배출 "B" CALL --> AMR
NOT
MOV       0 D072032	// 배출 "B" CALL --> AMR
; L135 (block mask: not executed)
LOAD      M04102	// PLT "B" 공정 자동 선택 중
AND       K04100	// PLT "B" Full 작업완료
AND       T4104	// PLT "B" 푸샤 전진완료
AND       T4107	// PLT "B" 락킹 풀림완료
MOV       1 D072033	// 배출 "B" 진입 요청 --> AMR
NOT
MOV       0 D072033	// 배출 "B" 진입 요청 --> AMR
; L137 (block mask: not executed)
LOAD      M04102	// PLT "B" 공정 자동 선택 중
AND       T4107	// PLT "B" 락킹 풀림완료
AND       M04120	// PLT "B" 파트 없음
AND NOT   T4105	// PLT "B" 푸샤 후진완료
MOV       1 D072034	// 배출 "B" 안착 완료 --> AMR
NOT
MOV       0 D072034	// 배출 "B" 안착 완료 --> AMR
; L139 (block mask: not executed)
LOAD      F00099
MOV       D004061 D072035	// OUT PLT "B" LOAD COMP 카운터 / 배출 "B" 소재 수량 ---> AMR

